// SIMATIC STEP 7 (V5.x) project CAN-O-MAT
// CPU: CPU 314C-2 DP
// station: P_ADR_BUS
// station: Hardware
// station: SIMATIC 300(1)
// program: S7 Program(1)

SYMBOL_TABLE
"FC2"	FC 2	FC 2	// Освещение внутри каномата
"FC3"	FC 3	FC 3	// Блок управления основным приводом
"FC4"	FC 4	FC 4	// Конвеер и подача корпусов
"FC6"	FC 6	FC 6	// Насос смазки (Опция)
"FC7"	FC 7	FC 7	// Смазка сужения
"1-А4"	I 14.1	BOOL	// Кнопки СТОП
"2-S19==2-S22"	I 14.2	BOOL	// Защитное устройство (окна)
"3-М1"	I 14.3	BOOL	// Основной привод включен
"7-Q7"	I 14.5	BOOL	// Автомат защиты насоса смазки банки
"8-Q8"	I 14.6	BOOL	// АВ защиты Кран(опция)
"10-М9а"	I 14.7	BOOL	// Транспорт подачи крышки включен
"РЕЗЕРВ 5"	I 15.0	BOOL	// Внешнее разрешение (или перемычка)
"РЕЗЕРВ 1"	I 15.1	BOOL	// Внешнее разрешение (или перемычка)
"Резерв"	I 15.2	BOOL	// Перемычка
"9-В34"	I 15.5	BOOL	// Опция
"9-В35Е==9-В35S"	I 15.6	BOOL	// Синхронизация выбрасывателя тестовой банки (опция)
"6-Q2"	I 15.7	BOOL	// Автомат защиты масляного насоса
"11-М10а"	I 16.4	BOOL	// Входной транспортер включен
"РЕЗЕРВ 2"	I 16.5	BOOL	// Резерв
"РЕЗЕРВ 3"	I 16.6	BOOL	// Резерв
"5-S11"	I 20.0	BOOL	// Автоматическая работа
"5-S29"	I 20.1	BOOL	// Jog Назад
"ET200S"	I 20.2	BOOL	// Питание подано
"5-S26"	I 20.3	BOOL	// Jog Вперед
"9-S10"	I 20.4	BOOL	// Сжатый воздух
"6-S1"	I 20.5	BOOL	// Давление масла за фильтром
"7-S27"	I 20.6	BOOL	// Наличие давления смазки
"7-S28"	I 20.7	BOOL	// Уровень смазки в бачке
"9-В28"	I 21.0	BOOL	// Датчик увеличения скорости каномата
"9-В29"	I 21.1	BOOL	// Наличие банки(входной конв)
"9-В30"	I 21.2	BOOL	// Датчик затора на выходном конвейере
"3-М1М"	I 21.3	BOOL	// Контроль температур Основного мотора
"9-В10"	I 21.4	BOOL	// Датчик такта
"9-В9"	I 21.5	BOOL	// Входящий запрос
"9-В27"	I 21.6	BOOL	// Опрос выхода
"9-В11"	I 21.7	BOOL	// Станция зауживания
"9-В12"	I 22.0	BOOL	// Станция отбортовки
"9-В13"	I 22.1	BOOL	// Станция зауживания
"9-В14"	I 22.2	BOOL	// Станция закатки №1
"9-В15"	I 22.3	BOOL	// Станция закатки №2
"6-S3"	I 22.6	BOOL	// Импульсы смазки (опция)
"11-B1"	I 22.7	BOOL	// Переполнение входного конвеера
"5-S230"	I 23.0	BOOL	// Кнопка СБРОС
"РЕЗЕРВ 4"	I 23.2	BOOL	// Резерв
"10-В29"	I 23.3	BOOL	// Такт подачи крышки
"10-В30"	I 23.4	BOOL	// Опрос крышки
"10-B31"	I 23.5	BOOL	// Наличие крышки на ленте
"10-В32"	I 23.6	BOOL	// Наличие крышки в магазине
"10-В33"	I 23.7	BOOL	// Наличие крышки
"5-S244"	I 24.4	BOOL	// Основной мотор ВКЛ
"5-S245"	I 24.5	BOOL	// Основной мотор ОТКЛ
"5-S246"	I 24.6	BOOL	// Каномат СТОП Открыт
"5-S247"	I 24.7	BOOL	// Каномат СТОП Закрыт
"М0.0"	M 0.0	BOOL	// Меркер всегда выключ.
"М0.1"	M 0.1	BOOL	// Теплый пуск CPU. Меркер всегда включен
"М0.5"	M 0.5	BOOL	// Меркер всегда выключ.
"М1.0"	M 1.0	BOOL	// Меркер неисправного состояния
"М1.1"	M 1.1	BOOL	// Тригер Основной мотор ВКЛ(Ручн. реж)
"М1.2"	M 1.2	BOOL	// Тригер Основной мотор ВКЛ(Авт. реж)
"М1.3"	M 1.3	BOOL	// Тригер Основной мотор Jog Вперед
"М1.5"	M 1.5	BOOL	// Тригер Основной мотор Jog Назад
"М2.0"	M 2.0	BOOL	// Меркер включения Основного мотора
"М2.2"	M 2.2	BOOL	// Входной конвейер переполнен
"М2.7"	M 2.7	BOOL	// Меркер затора на выходном конвейере
"М3.0"	M 3.0	BOOL	// Тригер включ. конвеера
"М3.3"	M 3.3	BOOL	// Наличие банки на входе
"М4.0"	M 4.0	BOOL	// Тригер включ. освещение каномата
"М6.2"	M 6.2	BOOL	// Меркер включ. масляного насоса для сужения
"М12.0"	M 12.0	BOOL	// Меркер включ. клапана подачи корпусов
"М16.4"	M 16.4	BOOL	// Меркер включения входного транспорт.
"М16.5"	M 16.5	BOOL	// Меркер включения РЕЗЕРВ 9
"М100.3"	M 100.3	BOOL	// Меркер ВКЛ входного транспорт
"М100.4"	M 100.4	BOOL	// РЕЗЕРВ 2,3 Всегда включен
"М100.7"	M 100.7	BOOL	// Входной транспорт. РАБОТАЕТ
"М101.0"	M 101.0	BOOL	// Меркер нормальной работы
"М220.1"	M 220.1	BOOL	// Автомат защиты насоса смазки банки ВЫКЛЮЧЕН
"М220.2"	M 220.2	BOOL	// АВ защиты Кран (опция) ВЫКЛЮЧЕН
"М221.0"	M 221.0	BOOL	// Нажата Аварийная кнопка СТОП
"М221.1"	M 221.1	BOOL	// Защитное устройство ОТКРЫТО
"М221.2"	M 221.2	BOOL	// Меркер контроля выкл. состояния Основного привода
"М221.3"	M 221.3	BOOL	// Меркер контроля температур Основного мотора
"М221.6"	M 221.6	BOOL	// НЕТ давления масла на сужении
"М222.0"	M 222.0	BOOL	// НЕТ крышки в магазине
"М222.3"	M 222.3	BOOL	// НЕТ смазки (опция)
"М222.5"	M 222.5	BOOL	// Синхронизация выбрасывателя тестовой банки (опция)
"М222.6"	M 222.6	BOOL	// Автомат защиты масляного насоса ВЫКЛЮЧЕН
"М223.5"	M 223.5	BOOL	// Каномат остановлен
"М223.7"	M 223.7	BOOL	// Транспорт подачи крышки ВЫКЛЮЧЕН
"М227.7"	M 227.7	BOOL	// Входной транспорт. НЕ РАБОТАЕТ
"М229.0"	M 229.0	BOOL	// Исправная работа
"М229.1"	M 229.1	BOOL	// Затор на выходном конвейере
"М248.2"	M 248.2	BOOL	// Меркер Освещение каномата Выключено
"М249.4"	M 249.4	BOOL	// Входной транспорт. ВЫКЛЮЧЕН
"М249.6"	M 249.6	BOOL	// РЕЗЕРВ 9 ВЫКЛЮЧЕН
"М250.2"	M 250.2	BOOL	// Меркер Освещение каномата Включено
"М251.4"	M 251.4	BOOL	// Входной транспорт. ВКЛЮЧЕН
"М251.6"	M 251.6	BOOL	// РЕЗЕРВ 9 ВКЛЮЧЕН
"3-К1"	Q 14.0	BOOL	// Подача питания на частотные привода
"1-К5"	Q 14.1	BOOL	// Сброс  Перезагрузка
"2-К3"	Q 14.2	BOOL	// Освещение каномата
"3-М1-2"	Q 14.3	BOOL	// Основной мотор (быстрое торможение
"3-M1-3"	Q 14.4	BOOL	// Основной мотор(Jog вперед)
"3-М1-4"	Q 14.5	BOOL	// Основной мотор(Jog назад)
"12-К2"	Q 14.6	BOOL	// Каномат в ожидании
"12-К3"	Q 14.7	BOOL	// Каномат в ожидании
"3-М1-1"	Q 15.0	BOOL	// Основной мотор (ВКЛ)
"12-К1"	Q 15.1	BOOL	// Каномат в работе
"7-K7"	Q 15.2	BOOL	// Масляной насос для сужения
"10-M9"	Q 15.4	BOOL	// Транспортер подачи крышки
"6-К2"	Q 15.5	BOOL	// Насос смазки (Опция)
"9-Y10"	Q 15.6	BOOL	// Опция
"11-М10"	Q 16.4	BOOL	// Входной транспортер
"РЕЗЕРВ 9"	Q 16.5	BOOL	// Резерв
"РЕЗЕРВ 10"	Q 16.6	BOOL	// Резерв
"РЕЗЕРВ 6"	Q 17.5	BOOL	// Резерв
"РЕЗЕРВ 7"	Q 17.6	BOOL	// Резерв
"РЕЗЕРВ 8"	Q 17.7	BOOL	// Резерв
"9-Y3"	Q 20.0	BOOL	// Клапан подачи корпусов
"7-Y5"	Q 20.1	BOOL	// Клапан распыления при сужении
"10-Y14"	Q 20.2	BOOL	// Клапан подачи крышки
"5-Н203"	Q 20.3	BOOL	// Лампа АВАРИЯ
"5-Н206"	Q 20.6	BOOL	// Лампа Основной мотор Включен
"5-Н207"	Q 20.7	BOOL	// Лампа Конвеер Включен
"SET_CLK"	SFC 0	SFC 0	// Set System Clock
"READ_CLK"	SFC 1	SFC 1	// Read System Clock
"SET_RTM"	SFC 2	SFC 2	// Set Run-Time Meter
"CTRL_RTM"	SFC 3	SFC 3	// Start/Stop Run-Time Meter
"READ_RTM"	SFC 4	SFC 4	// Read Run-Time Meter
"BLKMOV"	SFC 20	SFC 20	// Copy Variables
"FILL"	SFC 21	SFC 21	// Initialize a Memory Area
"Т1"	T 1	TIMER	// Задержка выключения 3-К1
"Т2"	T 2	TIMER	// Задержка срабатывания 9-В29 (включ.)
"Т3"	T 3	TIMER	// Таймер включ. на 1 сек. и выключ.
"Т4"	T 4	TIMER	// Задержка срабатывания 9-В29 (отключ.)
"Т11"	T 11	TIMER	// Задержка включения
"Т14"	T 14	TIMER	// Задержка срабатывания датчика 9-В28
"Т15"	T 15	TIMER	// Задержка включения датчика 9-В30 Затор на выходном конв
"Т16"	T 16	TIMER	// Задержка выключен датчика 9-В30 Затор на выходном конв.
"Т22"	T 22	TIMER	// Задержка включ. датчика 11-В1
"Т26"	T 26	TIMER	// Задержка включен. РЕЗЕРВ 5
"Т27"	T 27	TIMER	// Задержка выключен. РЕЗЕРВ 5
"Т28"	T 28	TIMER	// Задержка выключен. РЕЗЕРВ 1
"Т29"	T 29	TIMER	// Задержка включен. РЕЗЕРВ 1
"Т37"	T 37	TIMER	// Задержка отключения
"Т39"	T 39	TIMER	// Задержка включения
"Т40"	T 40	TIMER	// Задержка срабатывания
"Т42"	T 42	TIMER	// Задержка отключ. датчика 11-В1
"Т44"	T 44	TIMER	// Задержка включения "М0.1"
"Т45"	T 45	TIMER	// Таймер отсчитывает время и выключает
"Т46"	T 46	TIMER	// Задержка включения 2-S19=2S22
"Т50"	T 50	TIMER	// Таймер срабатыв. через время после начала тормож. Осн.  мотора
"Т52"	T 52	TIMER	// Задержка срабатыван датчика такта во включ. положении
"Т53"	T 53	TIMER	// Задержка срабатыван датчика такта в отключ. положении
"Т60"	T 60	TIMER	// Время смазки
"Т61"	T 61	TIMER	// Время между смазками
"Т120"	T 120	TIMER	// Задержка включ. клапана подачи корпусов
END_SYMBOL_TABLE

FUNCTION_BLOCK FB 100
AUTHOR : Joehring
VERSION : 0.1
BEGIN
// (block stored without names or comments; labels and parameter names are numbered)
NETWORK
TITLE =
      BLD   7;
      =     L 8.0;
      TAR2  LD 4;
      L     DINO;
      T     LW 9;
      +AR2  P#12.0;
      TAR2;
      LAR2  LD 4;
      T     LD 11;
      UC    "READ_CLK";
      {     P#L 2.0, P#L 9.0 };
      LAR2  LD 4;
      BLD   8;
      NOP   0;
NETWORK
TITLE =
      A(;
      A(;
      L     DIW [AR2,P#0.0];
      L     DIW [AR2,P#2.0];
      ==I;
      );
      =     L 0.0;
      A     L 0.0;
      FP    DIX [AR2,P#42.2];
      JNB   M001;
      L     DID 12;
      T     DID 24;
      SET;
      SAVE;
      CLR;
M001: A     BR;
      );
      JNB   M002;
      L     DID 16;
      T     DID 28;
M002: NOP   0;
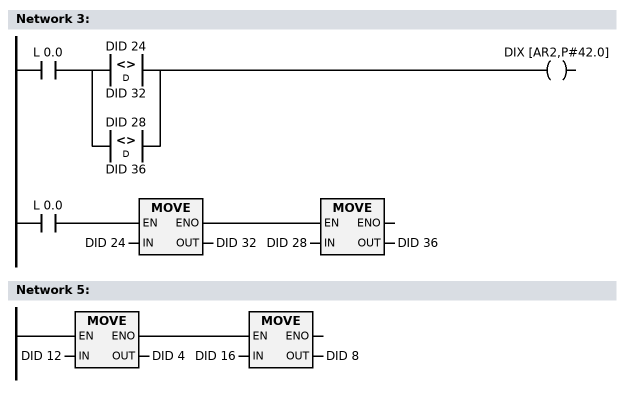
NETWORK
TITLE =
      A     L 0.0;
      =     L 4.0;
      A     L 4.0;
      A(;
      O(;
      L     DID 24;
      L     DID 32;
      <>D;
      );
      O(;
      L     DID 28;
      L     DID 36;
      <>D;
      );
      );
      =     DIX [AR2,P#42.0];
      A(;
      A     L 4.0;
      JNB   M003;
      L     DID 24;
      T     DID 32;
      SET;
      SAVE;
      CLR;
M003: A     BR;
      );
      JNB   M004;
      L     DID 28;
      T     DID 36;
M004: NOP   0;
NETWORK
TITLE =
      A     DIX [AR2,P#42.0];
      FP    DIX [AR2,P#42.1];
      JNB   M005;
      BLD   7;
      =     L 8.0;
      TAR2  LD 4;
      L     DINO;
      T     LW 9;
      +AR2  P#24.0;
      TAR2;
      LAR2  LD 4;
      T     LD 11;
      UC    "SET_CLK";
      {     P#L 9.0, P#L 2.0 };
      LAR2  LD 4;
      BLD   8;
M005: NOP   0;
NETWORK
TITLE =
      A(;
      L     DID 12;
      T     DID 4;
      SET;
      SAVE;
      CLR;
      A     BR;
      );
      JNB   M006;
      L     DID 16;
      T     DID 8;
M006: NOP   0;
END_FUNCTION_BLOCK

// FB 125: know-how protected block, not included

FUNCTION "FC2" : VOID	// FC 2
TITLE = Освещение внутри каномата.
//Включение освещения внутри каномата.
AUTHOR : Stolz
VERSION : 0.1
VAR_TEMP
  TEMP0 : BOOL ;
END_VAR
BEGIN
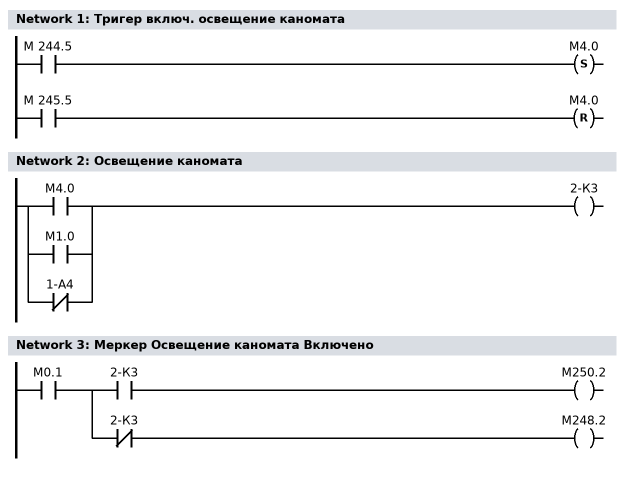
NETWORK
TITLE = Тригер включ. освещение каномата
      A     M 244.5;
      S     "М4.0";
      A     M 245.5;
      R     "М4.0";
      NOP   0;
NETWORK
TITLE = Освещение каномата
      O     "М4.0";
      O     "М1.0";
      ON    "1-А4";
      =     "2-К3";
NETWORK
TITLE = Меркер Освещение каномата Включено
      A     "М0.1";
      =     L 1.0;
      A     L 1.0;
      A     "2-К3";
      =     "М250.2";
      A     L 1.0;
      AN    "2-К3";
      =     "М248.2";
END_FUNCTION

FUNCTION "FC3" : VOID	// FC 3
TITLE = Блок управления основным приводом.
AUTHOR : Stolz
FAMILY : Maschfkt
NAME : Hauptmot
VERSION : 0.1
BEGIN
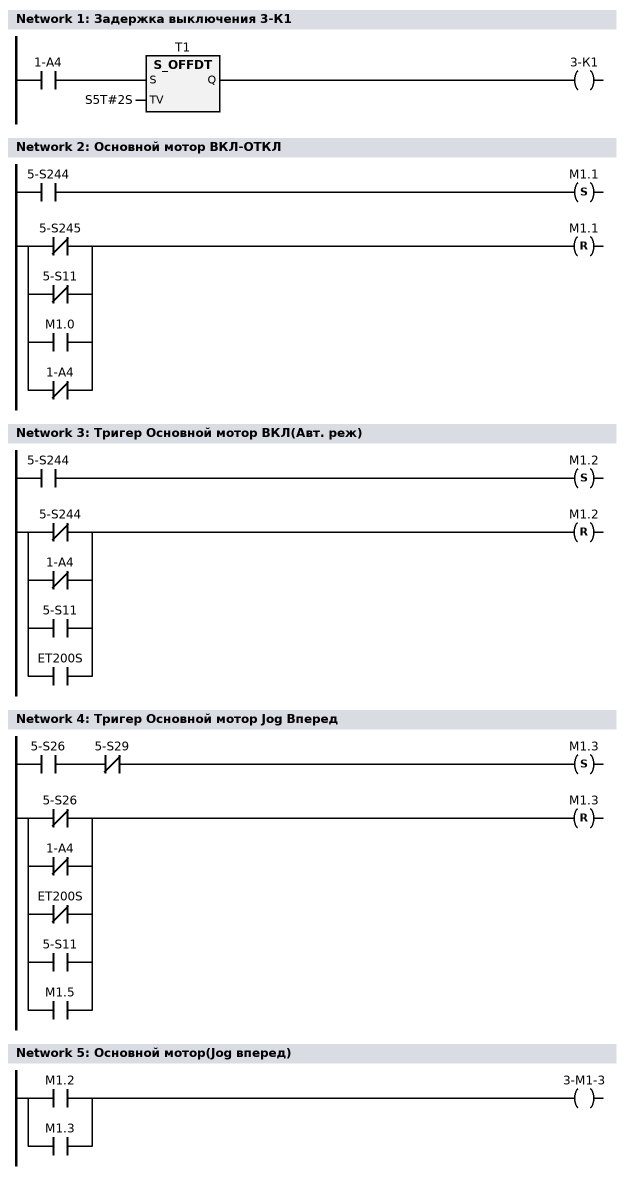
NETWORK
TITLE = Задержка выключения 3-К1
//После нажатия на любую из аварийных кнопок СТОП питание с частотных приводов 
//отключится спустя время, установленное в Т1.
      A     "1-А4";
      L     S5T#2S;
      SF    "Т1";
      NOP   0;
      NOP   0;
      NOP   0;
      A     "Т1";
      =     "3-К1";
NETWORK
TITLE = Основной мотор ВКЛ-ОТКЛ
      A     "5-S244";
      S     "М1.1";
      A(;
      ON    "5-S245";
      ON    "5-S11";
      O     "М1.0";
      ON    "1-А4";
      );
      R     "М1.1";
      NOP   0;
NETWORK
TITLE = Тригер Основной мотор ВКЛ(Авт. реж)
      A     "5-S244";
      S     "М1.2";
      A(;
      ON    "5-S244";
      ON    "1-А4";
      O     "5-S11";
      O     "ET200S";
      );
      R     "М1.2";
      NOP   0;
NETWORK
TITLE = Тригер Основной мотор Jog Вперед
      A     "5-S26";
      AN    "5-S29";
      S     "М1.3";
      A(;
      ON    "5-S26";
      ON    "1-А4";
      ON    "ET200S";
      O     "5-S11";
      O     "М1.5";
      );
      R     "М1.3";
      NOP   0;
NETWORK
TITLE = Основной мотор(Jog вперед)
      O     "М1.2";
      O     "М1.3";
      =     "3-M1-3";
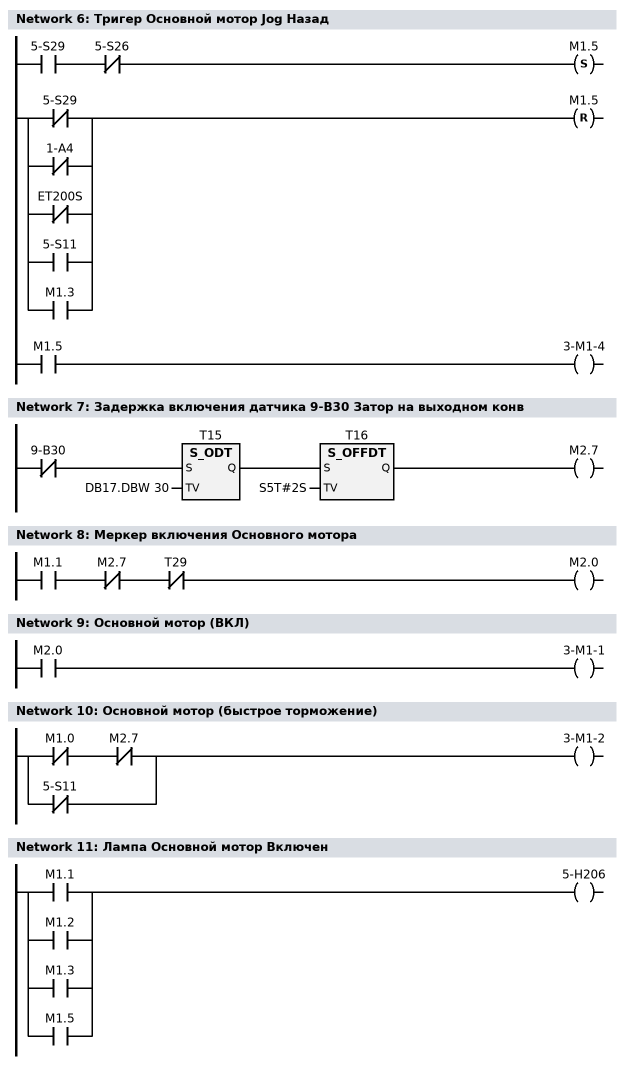
NETWORK
TITLE = Тригер Основной мотор Jog Назад
      A     "5-S29";
      AN    "5-S26";
      S     "М1.5";
      A(;
      ON    "5-S29";
      ON    "1-А4";
      ON    "ET200S";
      O     "5-S11";
      O     "М1.3";
      );
      R     "М1.5";
      A     "М1.5";
      =     "3-М1-4";
NETWORK
TITLE = Задержка включения датчика 9-В30 Затор на выходном конв
      A(;
      AN    "9-В30";
      L     DB17.DBW 30;
      SD    "Т15";
      NOP   0;
      NOP   0;
      NOP   0;
      A     "Т15";
      );
      L     S5T#2S;
      SF    "Т16";
      NOP   0;
      NOP   0;
      NOP   0;
      A     "Т16";
      =     "М2.7";
NETWORK
TITLE = Меркер включения Основного мотора
      A     "М1.1";
      AN    "М2.7";
      AN    "Т29";
      =     "М2.0";
NETWORK
TITLE = Основной мотор (ВКЛ)
      A     "М2.0";
      =     "3-М1-1";
NETWORK
TITLE = Основной мотор (быстрое торможение)
      AN    "М1.0";
      AN    "М2.7";
      ON    "5-S11";
      =     "3-М1-2";
NETWORK
TITLE = Лампа Основной мотор Включен
      O     "М1.1";
      O     "М1.2";
      O     "М1.3";
      O     "М1.5";
      =     "5-Н206";
END_FUNCTION

FUNCTION "FC4" : VOID	// FC 4
TITLE = Конвеер и подача корпусов.
AUTHOR : Stolz
VERSION : 0.1
VAR_TEMP
  TEMP0 : BOOL ;
END_VAR
BEGIN
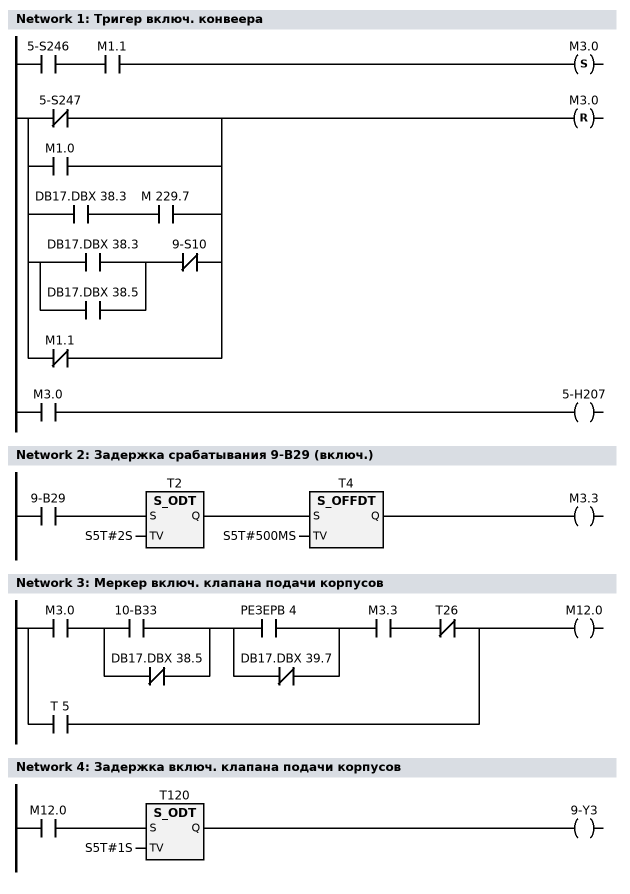
NETWORK
TITLE = Тригер включ. конвеера
      A     "5-S246";
      A     "М1.1";
      S     "М3.0";
      A(;
      ON    "5-S247";
      O     "М1.0";
      O;
      A     DB17.DBX 38.3;
      A     M 229.7;
      O;
      A(;
      O     DB17.DBX 38.3;
      O     DB17.DBX 38.5;
      );
      AN    "9-S10";
      ON    "М1.1";
      );
      R     "М3.0";
      A     "М3.0";
      =     "5-Н207";
NETWORK
TITLE = Задержка срабатывания 9-В29 (включ.)
      A(;
      A     "9-В29";
      L     S5T#2S;
      SD    "Т2";
      NOP   0;
      NOP   0;
      NOP   0;
      A     "Т2";
      );
      L     S5T#500MS;
      SF    "Т4";
      NOP   0;
      NOP   0;
      NOP   0;
      A     "Т4";
      =     "М3.3";
NETWORK
TITLE = Меркер включ. клапана подачи корпусов
      A     "М3.0";
      A(;
      O     "10-В33";
      ON    DB17.DBX 38.5;
      );
      A(;
      O     "РЕЗЕРВ 4";
      ON    DB17.DBX 39.7;
      );
      A     "М3.3";
      AN    "Т26";
      O     T 5;
      =     "М12.0";
NETWORK
TITLE = Задержка включ. клапана подачи корпусов
      A     "М12.0";
      L     S5T#1S;
      SD    "Т120";
      NOP   0;
      NOP   0;
      NOP   0;
      A     "Т120";
      =     "9-Y3";
END_FUNCTION

FUNCTION "FC6" : VOID	// FC 6
TITLE = Включение насоса смазки.
//Включение насоса смазки(Опция)
AUTHOR : Stolz
NAME : Schmier
VERSION : 0.1
BEGIN
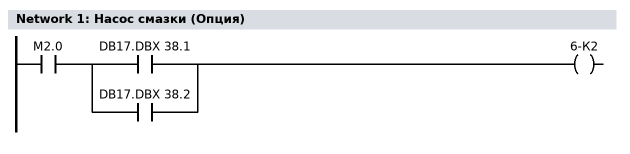
NETWORK
TITLE = Насос смазки (Опция)
      A     "М2.0";
      A(;
      O     DB17.DBX 38.1;
      O     DB17.DBX 38.2;
      );
      =     "6-К2";
END_FUNCTION

FUNCTION "FC7" : VOID	// FC 7
TITLE = Блок управления смазкой сужения.
AUTHOR : Stolz
VERSION : 0.1
BEGIN
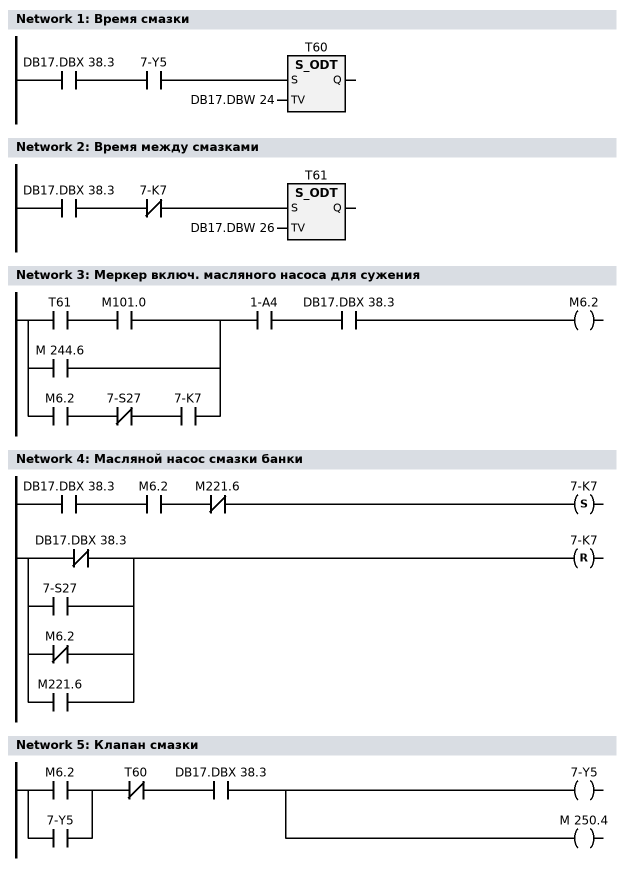
NETWORK
TITLE = Время смазки
      A     DB17.DBX 38.3;
      A     "7-Y5";
      L     DB17.DBW 24;
      SD    "Т60";
      NOP   0;
      NOP   0;
      NOP   0;
      NOP   0;
NETWORK
TITLE = Время между смазками
      A     DB17.DBX 38.3;
      AN    "7-K7";
      L     DB17.DBW 26;
      SD    "Т61";
      NOP   0;
      NOP   0;
      NOP   0;
      NOP   0;
NETWORK
TITLE = Меркер включ. масляного насоса для сужения
      A(;
      A     "Т61";
      A     "М101.0";
      O     M 244.6;
      O;
      A     "М6.2";
      AN    "7-S27";
      A     "7-K7";
      );
      A     "1-А4";
      A     DB17.DBX 38.3;
      =     "М6.2";
NETWORK
TITLE = Масляной насос смазки банки
      A     DB17.DBX 38.3;
      A     "М6.2";
      AN    "М221.6";
      S     "7-K7";
      A(;
      ON    DB17.DBX 38.3;
      O     "7-S27";
      ON    "М6.2";
      O     "М221.6";
      );
      R     "7-K7";
      NOP   0;
NETWORK
TITLE = Клапан смазки
      A(;
      O     "М6.2";
      O     "7-Y5";
      );
      AN    "Т60";
      A     DB17.DBX 38.3;
      =     "7-Y5";
      =     M 250.4;
END_FUNCTION

FUNCTION FC 10 : VOID
AUTHOR : Stolz
NAME : Deckelfi
VERSION : 0.3
VAR_TEMP
  TEMP0 : DWORD ;
  TEMP1 : BOOL ;
  TEMP2 : BOOL ;
  TEMP3 : BOOL ;
END_VAR
BEGIN
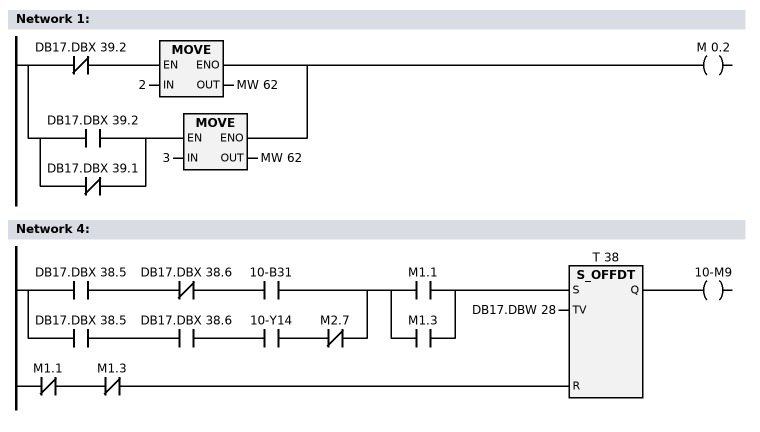
NETWORK
TITLE =
      O(;
      AN    DB17.DBX 39.2;
      JNB   _001;
      L     2;
      T     MW 62;
      SET;
      SAVE;
      CLR;
_001: A     BR;
      );
      O(;
      A(;
      O     DB17.DBX 39.2;
      ON    DB17.DBX 39.1;
      );
      JNB   _002;
      L     3;
      T     MW 62;
      SET;
      SAVE;
      CLR;
_002: A     BR;
      );
      =     M 0.2;
NETWORK
TITLE =
      A(;
      A     M 21.4;
      CD    C 36;
      BLD   101;
      A(;
      O     M 21.7;
      O     "5-S246";
      );
      L     MW 62;
      S     C 36;
      NOP   0;
      NOP   0;
      NOP   0;
      A     C 36;
      );
      NOT;
      =     #TEMP1;
NETWORK
TITLE =
      A(;
      A     M 21.7;
      CD    C 37;
      BLD   101;
      A(;
      O     #TEMP1;
      O     "5-S246";
      );
      L     DB17.DBW 56;
      S     C 37;
      NOP   0;
      NOP   0;
      NOP   0;
      A     C 37;
      );
      NOT;
      A     "9-Y3";
      =     M 1.4;
NETWORK
TITLE =
      A(;
      A     DB17.DBX 38.5;
      AN    DB17.DBX 38.6;
      A     "10-B31";
      O;
      A     DB17.DBX 38.5;
      A     DB17.DBX 38.6;
      A     "10-Y14";
      AN    "М2.7";
      );
      A(;
      O     "М1.1";
      O     "М1.3";
      );
      L     DB17.DBW 28;
      SF    T 38;
      AN    "М1.1";
      AN    "М1.3";
      R     T 38;
      NOP   0;
      NOP   0;
      A     T 38;
      =     "10-M9";
END_FUNCTION

FUNCTION FC 11 : VOID
AUTHOR : Stolz
VERSION : 0.2
BEGIN
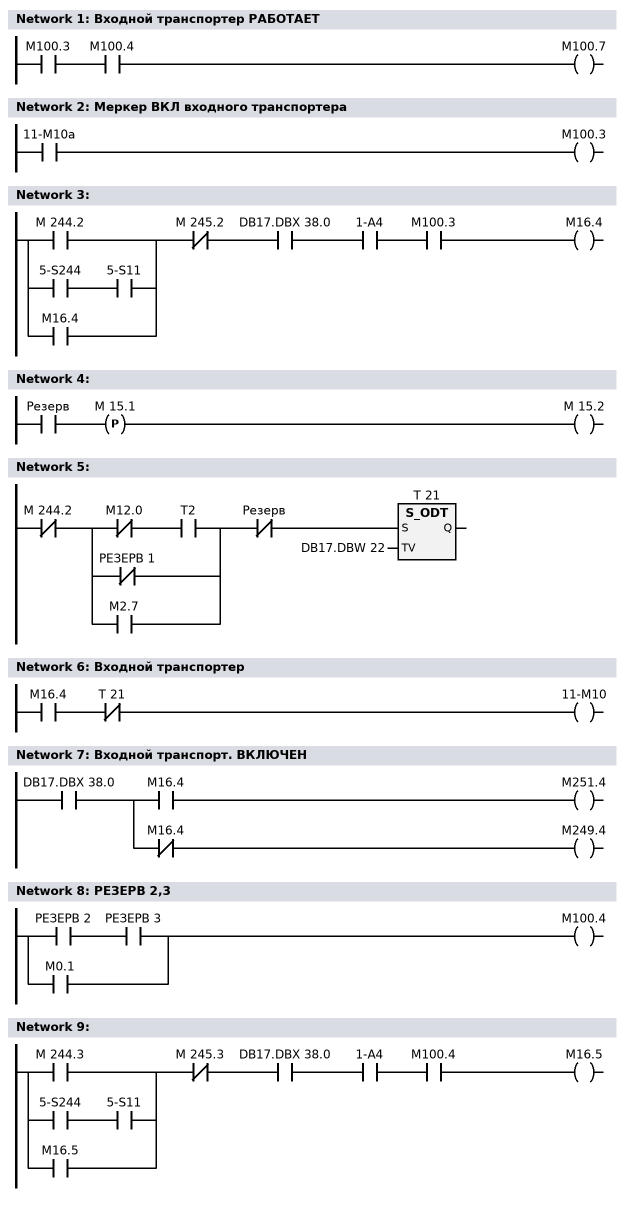
NETWORK
TITLE = Входной транспортер РАБОТАЕТ
      A     "М100.3";
      A     "М100.4";
      =     "М100.7";
NETWORK
TITLE = Меркер ВКЛ входного транспортера
      A     "11-М10а";
      =     "М100.3";
NETWORK
TITLE =
      A(;
      O     M 244.2;
      O;
      A     "5-S244";
      A     "5-S11";
      O     "М16.4";
      );
      AN    M 245.2;
      A     DB17.DBX 38.0;
      A     "1-А4";
      A     "М100.3";
      =     "М16.4";
NETWORK
TITLE =
      A     "Резерв";
      FP    M 15.1;
      =     M 15.2;
NETWORK
TITLE =
      AN    M 244.2;
      A(;
      AN    "М12.0";
      A     "Т2";
      ON    "РЕЗЕРВ 1";
      O     "М2.7";
      );
      AN    "Резерв";
      L     DB17.DBW 22;
      SD    T 21;
      NOP   0;
      NOP   0;
      NOP   0;
      NOP   0;
NETWORK
TITLE = Входной транспортер
      A     "М16.4";
      AN    T 21;
      =     "11-М10";
NETWORK
TITLE = Входной транспорт. ВКЛЮЧЕН
      A     DB17.DBX 38.0;
      =     L 0.0;
      A     L 0.0;
      A     "М16.4";
      =     "М251.4";
      A     L 0.0;
      AN    "М16.4";
      =     "М249.4";
NETWORK
TITLE = РЕЗЕРВ 2,3
      A     "РЕЗЕРВ 2";
      A     "РЕЗЕРВ 3";
      O     "М0.1";
      =     "М100.4";
NETWORK
TITLE =
      A(;
      O     M 244.3;
      O;
      A     "5-S244";
      A     "5-S11";
      O     "М16.5";
      );
      AN    M 245.3;
      A     DB17.DBX 38.0;
      A     "1-А4";
      A     "М100.4";
      =     "М16.5";
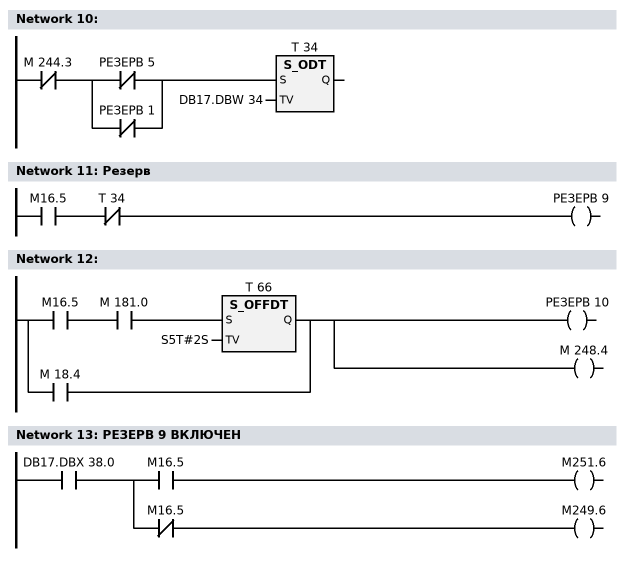
NETWORK
TITLE =
      AN    M 244.3;
      A(;
      ON    "РЕЗЕРВ 5";
      ON    "РЕЗЕРВ 1";
      );
      L     DB17.DBW 34;
      SD    T 34;
      NOP   0;
      NOP   0;
      NOP   0;
      NOP   0;
NETWORK
TITLE = Резерв
      A     "М16.5";
      AN    T 34;
      =     "РЕЗЕРВ 9";
NETWORK
TITLE =
      O(;
      A     "М16.5";
      A     M 181.0;
      L     S5T#2S;
      SF    T 66;
      NOP   0;
      NOP   0;
      NOP   0;
      A     T 66;
      );
      O     M 18.4;
      =     "РЕЗЕРВ 10";
      =     M 248.4;
NETWORK
TITLE = РЕЗЕРВ 9 ВКЛЮЧЕН
      A     DB17.DBX 38.0;
      =     L 0.0;
      A     L 0.0;
      A     "М16.5";
      =     "М251.6";
      A     L 0.0;
      AN    "М16.5";
      =     "М249.6";
END_FUNCTION

FUNCTION FC 12 : VOID
AUTHOR : Stolz
VERSION : 0.3
VAR_TEMP
  TEMP0 : DWORD ;
END_VAR
BEGIN
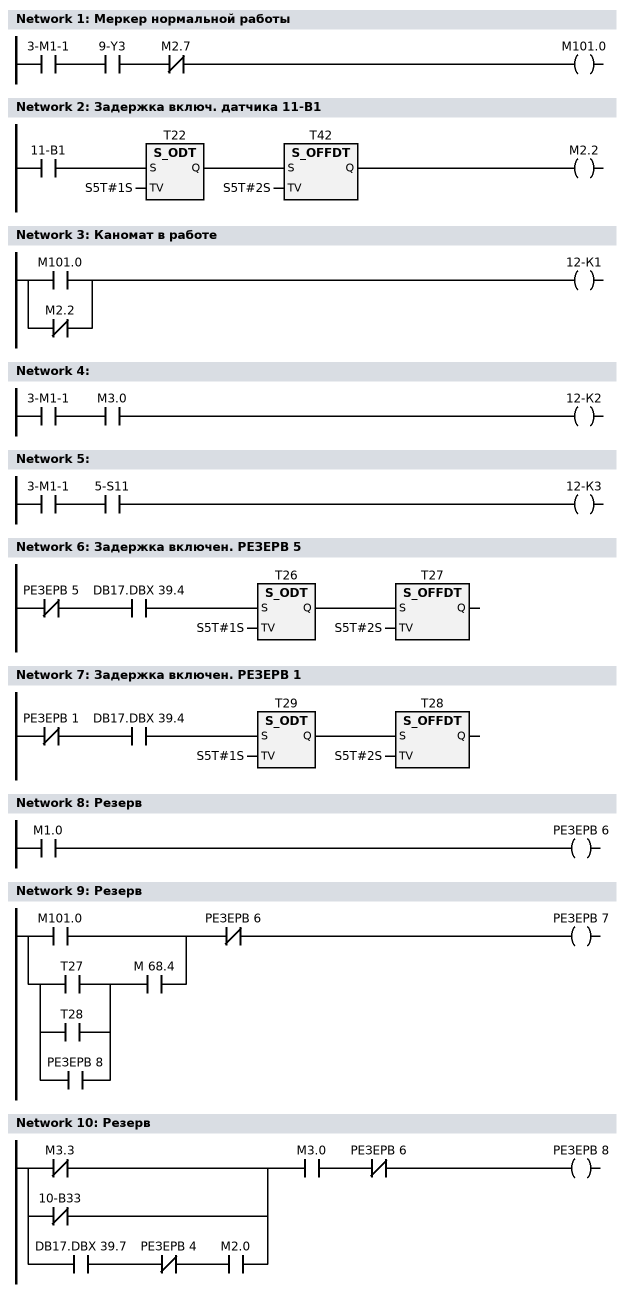
NETWORK
TITLE = Меркер нормальной работы
//Корпуса идут, банка на выходе идет нормально.
      A     "3-М1-1";
      A     "9-Y3";
      AN    "М2.7";
      =     "М101.0";
NETWORK
TITLE = Задержка включ. датчика 11-В1
      A(;
      A     "11-B1";
      L     S5T#1S;
      SD    "Т22";
      NOP   0;
      NOP   0;
      NOP   0;
      A     "Т22";
      );
      L     S5T#2S;
      SF    "Т42";
      NOP   0;
      NOP   0;
      NOP   0;
      A     "Т42";
      =     "М2.2";
NETWORK
TITLE = Каномат в работе
      O     "М101.0";
      ON    "М2.2";
      =     "12-К1";
NETWORK
TITLE =
      A     "3-М1-1";
      A     "М3.0";
      =     "12-К2";
NETWORK
TITLE =
      A     "3-М1-1";
      A     "5-S11";
      =     "12-К3";
NETWORK
TITLE = Задержка включен. РЕЗЕРВ 5
      A(;
      AN    "РЕЗЕРВ 5";
      A     DB17.DBX 39.4;
      L     S5T#1S;
      SD    "Т26";
      NOP   0;
      NOP   0;
      NOP   0;
      A     "Т26";
      );
      L     S5T#2S;
      SF    "Т27";
      NOP   0;
      NOP   0;
      NOP   0;
      NOP   0;
NETWORK
TITLE = Задержка включен. РЕЗЕРВ 1
      A(;
      AN    "РЕЗЕРВ 1";
      A     DB17.DBX 39.4;
      L     S5T#1S;
      SD    "Т29";
      NOP   0;
      NOP   0;
      NOP   0;
      A     "Т29";
      );
      L     S5T#2S;
      SF    "Т28";
      NOP   0;
      NOP   0;
      NOP   0;
      NOP   0;
NETWORK
TITLE = Резерв
      A     "М1.0";
      =     "РЕЗЕРВ 6";
NETWORK
TITLE = Резерв
      A(;
      O     "М101.0";
      O;
      A(;
      O     "Т27";
      O     "Т28";
      O     "РЕЗЕРВ 8";
      );
      A     M 68.4;
      );
      AN    "РЕЗЕРВ 6";
      =     "РЕЗЕРВ 7";
NETWORK
TITLE = Резерв
      A(;
      ON    "М3.3";
      ON    "10-В33";
      O;
      A     DB17.DBX 39.7;
      AN    "РЕЗЕРВ 4";
      A     "М2.0";
      );
      A     "М3.0";
      AN    "РЕЗЕРВ 6";
      =     "РЕЗЕРВ 8";
END_FUNCTION

FUNCTION FC 23 : VOID
AUTHOR : Stolz
VERSION : 0.2
VAR_TEMP
  TEMP0 : DINT ;
  TEMP1 : DINT ;
  TEMP2 : BOOL ;
  TEMP3 : BOOL ;
  TEMP4 : BOOL ;
  TEMP5 : BOOL ;
END_VAR
BEGIN
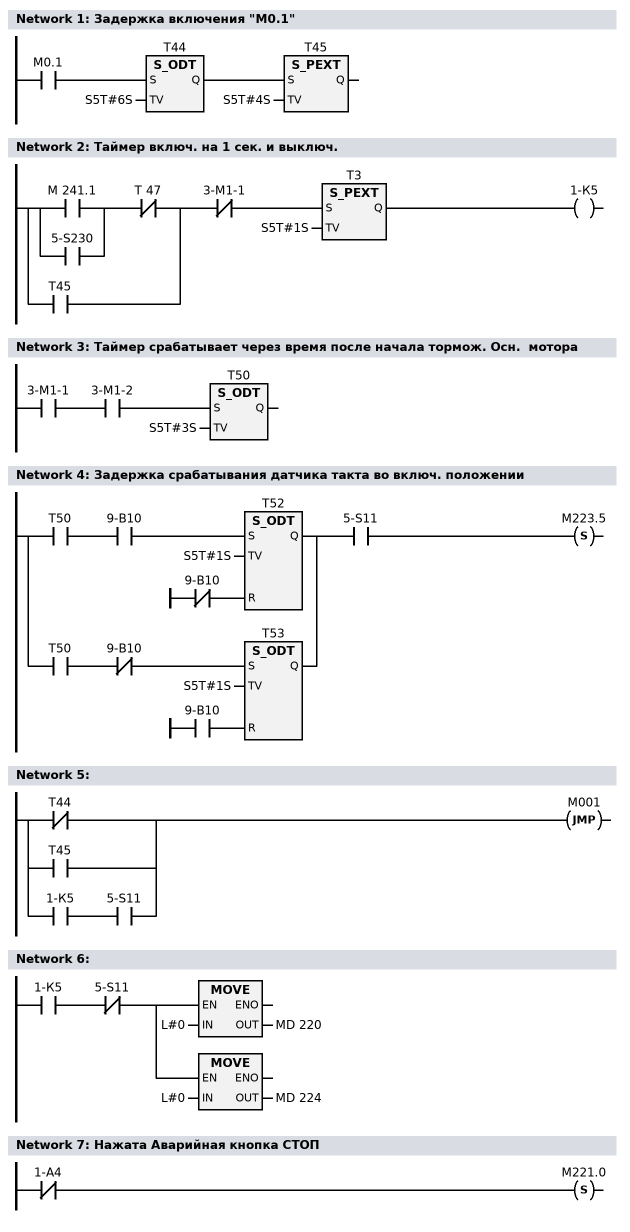
NETWORK
TITLE = Задержка включения "М0.1"
//Т44 включается через 6 сек. после подачи питания на каномат, Т45 включается 
//сразу после срабатывания Т44 и выключается через 4 сек. Остается выключенным до 
//конца работы.
      A(;
      A     "М0.1";
      L     S5T#6S;
      SD    "Т44";
      NOP   0;
      NOP   0;
      NOP   0;
      A     "Т44";
      );
      L     S5T#4S;
      SE    "Т45";
      NOP   0;
      NOP   0;
      NOP   0;
      NOP   0;
NETWORK
TITLE = Таймер включ. на 1 сек. и выключ.
      A(;
      A(;
      O     M 241.1;
      O     "5-S230";
      );
      AN    T 47;
      O     "Т45";
      );
      AN    "3-М1-1";
      L     S5T#1S;
      SE    "Т3";
      NOP   0;
      NOP   0;
      NOP   0;
      A     "Т3";
      =     "1-К5";
NETWORK
TITLE = Таймер срабатывает через время после начала тормож. Осн.  мотора
      A     "3-М1-1";
      A     "3-М1-2";
      L     S5T#3S;
      SD    "Т50";
      NOP   0;
      NOP   0;
      NOP   0;
      NOP   0;
NETWORK
TITLE = Задержка срабатывания датчика такта во включ. положении
      A(;
      O(;
      A     "Т50";
      A     "9-В10";
      L     S5T#1S;
      SD    "Т52";
      AN    "9-В10";
      R     "Т52";
      NOP   0;
      NOP   0;
      A     "Т52";
      );
      O(;
      A     "Т50";
      AN    "9-В10";
      L     S5T#1S;
      SD    "Т53";
      A     "9-В10";
      R     "Т53";
      NOP   0;
      NOP   0;
      A     "Т53";
      );
      );
      A     "5-S11";
      S     "М223.5";
NETWORK
TITLE =
      ON    "Т44";
      O     "Т45";
      O;
      A     "1-К5";
      A     "5-S11";
      JC    M001;
NETWORK
TITLE =
      A     "1-К5";
      AN    "5-S11";
      =     L 9.0;
      A     L 9.0;
      JNB   _001;
      L     L#0;
      T     MD 220;
_001: NOP   0;
      A     L 9.0;
      JNB   _002;
      L     L#0;
      T     MD 224;
_002: NOP   0;
NETWORK
TITLE = Нажата Аварийная кнопка СТОП
      AN    "1-А4";
      S     "М221.0";
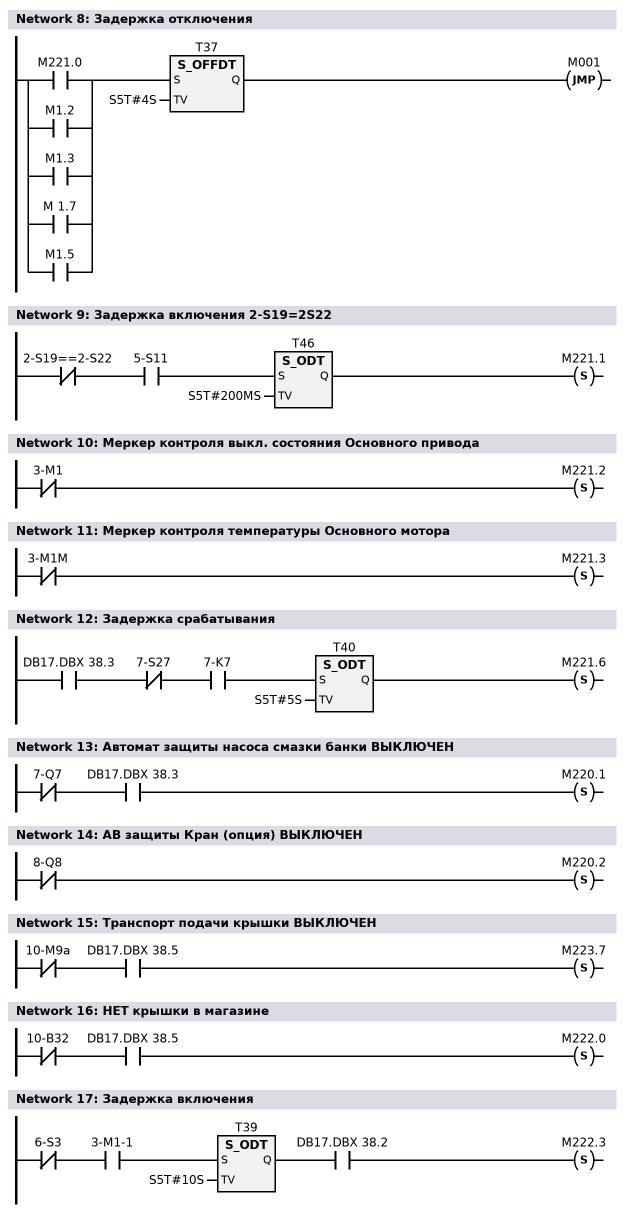
NETWORK
TITLE = Задержка отключения
      A(;
      O     "М221.0";
      O     "М1.2";
      O     "М1.3";
      O     M 1.7;
      O     "М1.5";
      );
      L     S5T#4S;
      SF    "Т37";
      NOP   0;
      NOP   0;
      NOP   0;
      A     "Т37";
      JC    M001;
NETWORK
TITLE = Задержка включения 2-S19=2S22
      AN    "2-S19==2-S22";
      A     "5-S11";
      L     S5T#200MS;
      SD    "Т46";
      NOP   0;
      NOP   0;
      NOP   0;
      A     "Т46";
      S     "М221.1";
NETWORK
TITLE = Меркер контроля выкл. состояния Основного привода
      AN    "3-М1";
      S     "М221.2";
NETWORK
TITLE = Меркер контроля температуры Основного мотора
      AN    "3-М1М";
      S     "М221.3";
NETWORK
TITLE = Задержка срабатывания
      A     DB17.DBX 38.3;
      AN    "7-S27";
      A     "7-K7";
      L     S5T#5S;
      SD    "Т40";
      NOP   0;
      NOP   0;
      NOP   0;
      A     "Т40";
      S     "М221.6";
NETWORK
TITLE = Автомат защиты насоса смазки банки ВЫКЛЮЧЕН
      AN    "7-Q7";
      A     DB17.DBX 38.3;
      S     "М220.1";
NETWORK
TITLE = АВ защиты Кран (опция) ВЫКЛЮЧЕН
      AN    "8-Q8";
      S     "М220.2";
NETWORK
TITLE = Транспорт подачи крышки ВЫКЛЮЧЕН
      AN    "10-М9а";
      A     DB17.DBX 38.5;
      S     "М223.7";
NETWORK
TITLE = НЕТ крышки в магазине
      AN    "10-В32";
      A     DB17.DBX 38.5;
      S     "М222.0";
NETWORK
TITLE = Задержка включения
      A(;
      AN    "6-S3";
      A     "3-М1-1";
      L     S5T#10S;
      SD    "Т39";
      NOP   0;
      NOP   0;
      NOP   0;
      A     "Т39";
      );
      A     DB17.DBX 38.2;
      S     "М222.3";
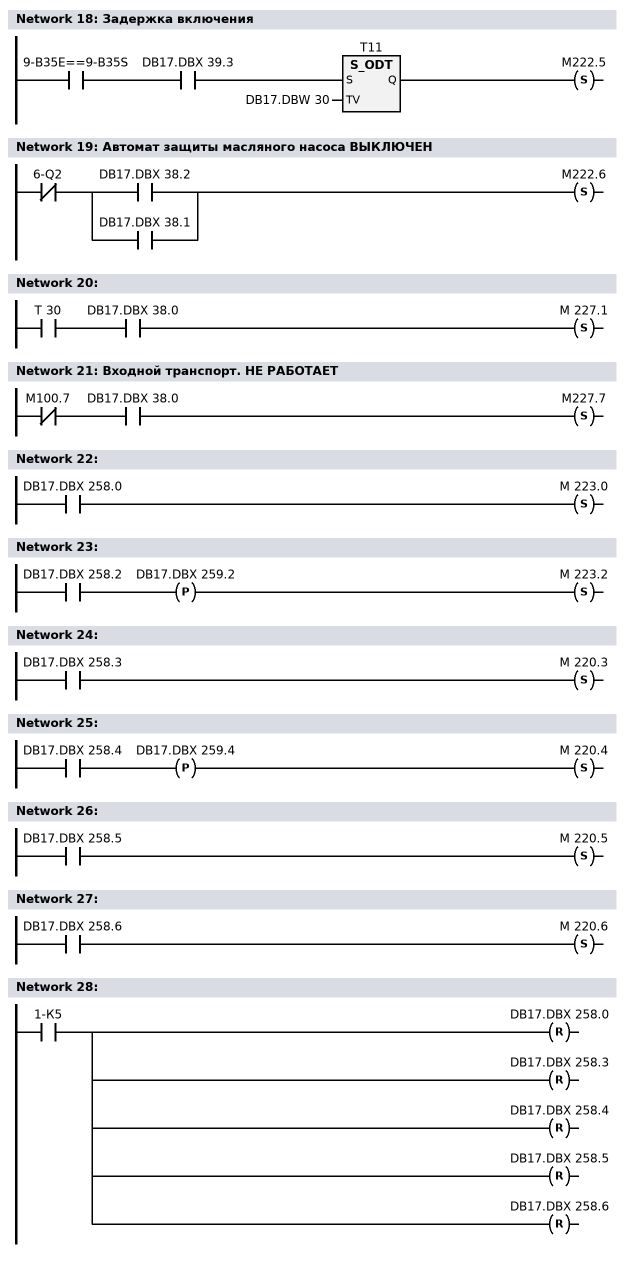
NETWORK
TITLE = Задержка включения
      A     "9-В35Е==9-В35S";
      A     DB17.DBX 39.3;
      L     DB17.DBW 30;
      SD    "Т11";
      NOP   0;
      NOP   0;
      NOP   0;
      A     "Т11";
      S     "М222.5";
NETWORK
TITLE = Автомат защиты масляного насоса ВЫКЛЮЧЕН
      AN    "6-Q2";
      A(;
      O     DB17.DBX 38.2;
      O     DB17.DBX 38.1;
      );
      S     "М222.6";
NETWORK
TITLE =
      A     T 30;
      A     DB17.DBX 38.0;
      S     M 227.1;
NETWORK
TITLE = Входной транспорт. НЕ РАБОТАЕТ
      AN    "М100.7";
      A     DB17.DBX 38.0;
      S     "М227.7";
NETWORK
TITLE =
      A     DB17.DBX 258.0;
      S     M 223.0;
NETWORK
TITLE =
      A     DB17.DBX 258.2;
      FP    DB17.DBX 259.2;
      S     M 223.2;
NETWORK
TITLE =
      A     DB17.DBX 258.3;
      S     M 220.3;
NETWORK
TITLE =
      A     DB17.DBX 258.4;
      FP    DB17.DBX 259.4;
      S     M 220.4;
NETWORK
TITLE =
      A     DB17.DBX 258.5;
      S     M 220.5;
NETWORK
TITLE =
      A     DB17.DBX 258.6;
      S     M 220.6;
NETWORK
TITLE =
      A     "1-К5";
      R     DB17.DBX 258.0;
      R     DB17.DBX 258.3;
      R     DB17.DBX 258.4;
      R     DB17.DBX 258.5;
      R     DB17.DBX 258.6;
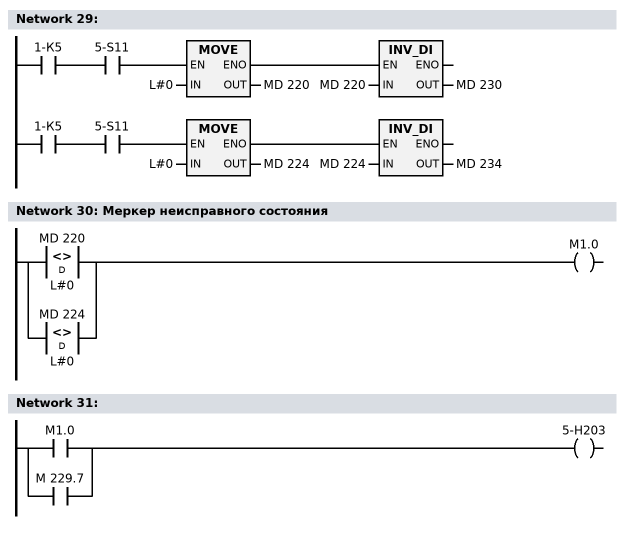
NETWORK
TITLE =
M001: A     "1-К5";
      A     "5-S11";
      =     L 9.0;
      A(;
      A     L 9.0;
      JNB   _003;
      L     L#0;
      T     MD 220;
      SET;
      SAVE;
      CLR;
_003: A     BR;
      );
      JNB   _004;
      L     MD 220;
      INVD;
      T     MD 230;
_004: NOP   0;
      A(;
      A     L 9.0;
      JNB   _005;
      L     L#0;
      T     MD 224;
      SET;
      SAVE;
      CLR;
_005: A     BR;
      );
      JNB   _006;
      L     MD 224;
      INVD;
      T     MD 234;
_006: NOP   0;
NETWORK
TITLE = Меркер неисправного состояния
      O(;
      L     MD 220;
      L     L#0;
      <>D;
      );
      O(;
      L     MD 224;
      L     L#0;
      <>D;
      );
      =     "М1.0";
NETWORK
TITLE =
      O     "М1.0";
      O     M 229.7;
      =     "5-Н203";
END_FUNCTION

FUNCTION FC 24 : VOID
AUTHOR : Stolz
VERSION : 0.2
BEGIN
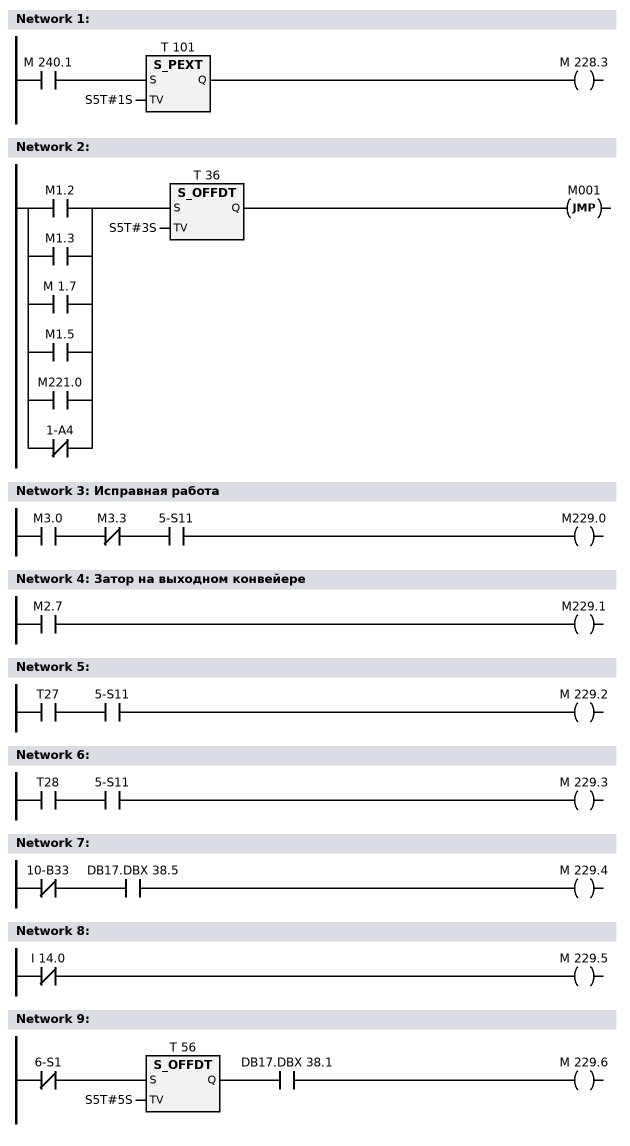
NETWORK
TITLE =
      A     M 240.1;
      L     S5T#1S;
      SE    T 101;
      NOP   0;
      NOP   0;
      NOP   0;
      A     T 101;
      =     M 228.3;
NETWORK
TITLE =
      A(;
      O     "М1.2";
      O     "М1.3";
      O     M 1.7;
      O     "М1.5";
      O     "М221.0";
      ON    "1-А4";
      );
      L     S5T#3S;
      SF    T 36;
      NOP   0;
      NOP   0;
      NOP   0;
      A     T 36;
      JC    M001;
NETWORK
TITLE = Исправная работа
      A     "М3.0";
      AN    "М3.3";
      A     "5-S11";
      =     "М229.0";
NETWORK
TITLE = Затор на выходном конвейере
      A     "М2.7";
      =     "М229.1";
NETWORK
TITLE =
      A     "Т27";
      A     "5-S11";
      =     M 229.2;
NETWORK
TITLE =
      A     "Т28";
      A     "5-S11";
      =     M 229.3;
NETWORK
TITLE =
      AN    "10-В33";
      A     DB17.DBX 38.5;
      =     M 229.4;
NETWORK
TITLE =
      AN    I 14.0;
      =     M 229.5;
NETWORK
TITLE =
      A(;
      AN    "6-S1";
      L     S5T#5S;
      SF    T 56;
      NOP   0;
      NOP   0;
      NOP   0;
      A     T 56;
      );
      A     DB17.DBX 38.1;
      =     M 229.6;
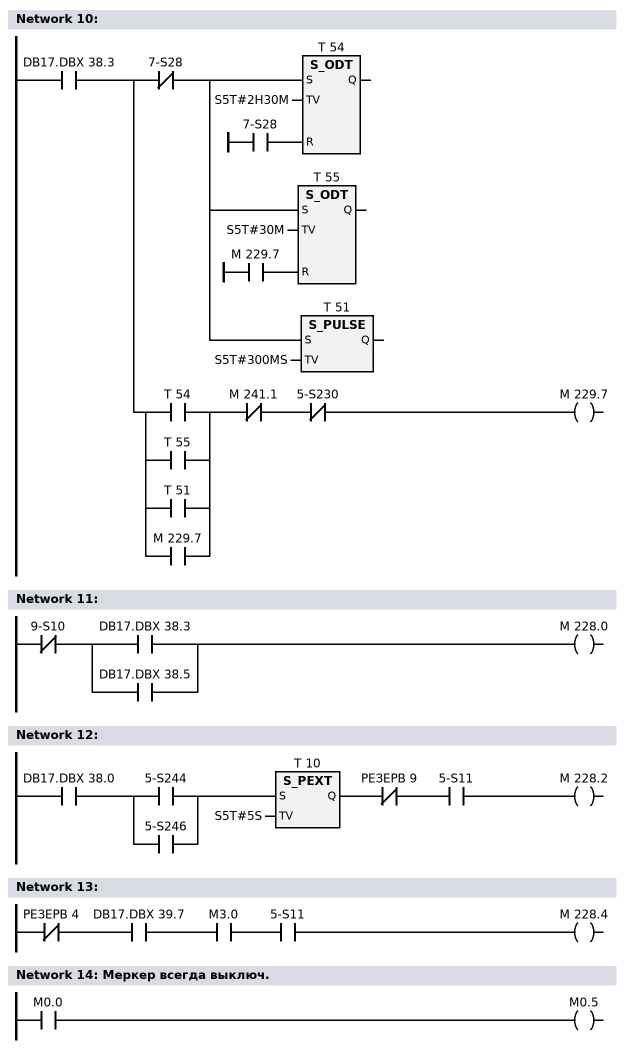
NETWORK
TITLE =
      A     DB17.DBX 38.3;
      =     L 0.0;
      A     L 0.0;
      AN    "7-S28";
      =     L 0.1;
      A     L 0.1;
      L     S5T#2H30M;
      SD    T 54;
      A     "7-S28";
      R     T 54;
      NOP   0;
      NOP   0;
      NOP   0;
      A     L 0.1;
      L     S5T#30M;
      SD    T 55;
      A     M 229.7;
      R     T 55;
      NOP   0;
      NOP   0;
      NOP   0;
      A     L 0.1;
      L     S5T#300MS;
      SP    T 51;
      NOP   0;
      NOP   0;
      NOP   0;
      NOP   0;
      A     L 0.0;
      A(;
      O     T 54;
      O     T 55;
      O     T 51;
      O     M 229.7;
      );
      AN    M 241.1;
      AN    "5-S230";
      =     M 229.7;
NETWORK
TITLE =
      AN    "9-S10";
      A(;
      O     DB17.DBX 38.3;
      O     DB17.DBX 38.5;
      );
      =     M 228.0;
NETWORK
TITLE =
      A(;
      A     DB17.DBX 38.0;
      A(;
      O     "5-S244";
      O     "5-S246";
      );
      L     S5T#5S;
      SE    T 10;
      NOP   0;
      NOP   0;
      NOP   0;
      A     T 10;
      );
      AN    "РЕЗЕРВ 9";
      A     "5-S11";
      =     M 228.2;
NETWORK
TITLE =
      AN    "РЕЗЕРВ 4";
      A     DB17.DBX 39.7;
      A     "М3.0";
      A     "5-S11";
      =     M 228.4;
NETWORK
TITLE = Меркер всегда выключ.
M001: A     "М0.0";
      =     "М0.5";
END_FUNCTION

FUNCTION FC 50 : VOID
AUTHOR : Stolz
VERSION : 0.2
BEGIN
// (block stored without names or comments; labels and parameter names are numbered)
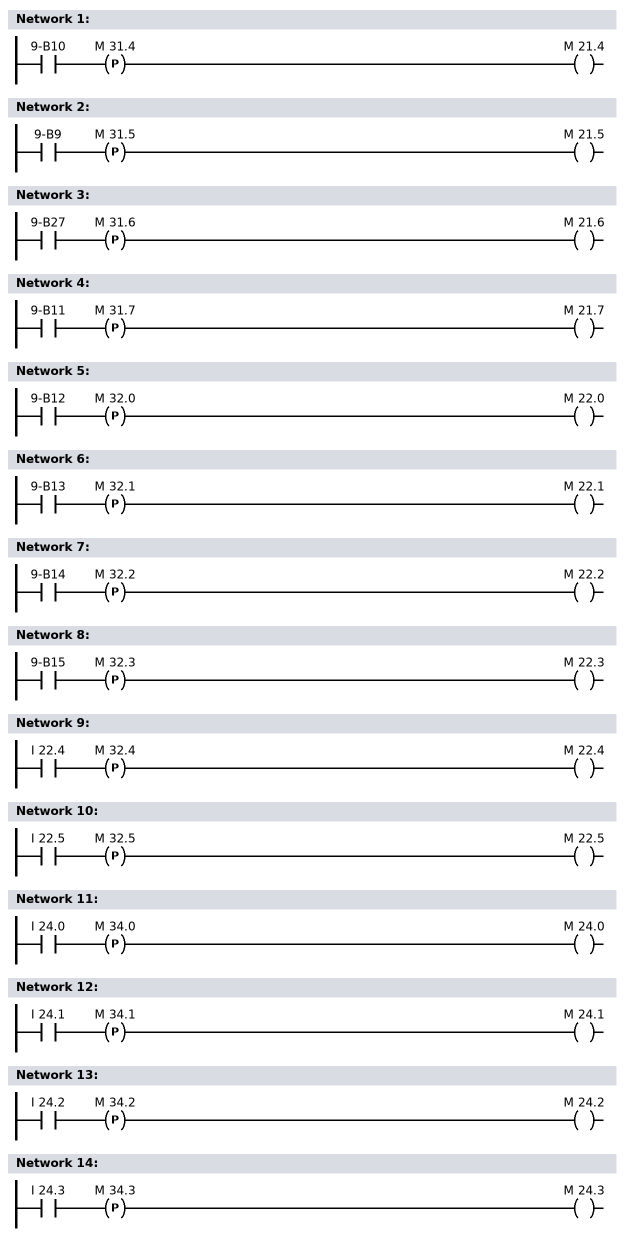
NETWORK
TITLE =
      A     "9-В10";
      FP    M 31.4;
      =     M 21.4;
NETWORK
TITLE =
      A     "9-В9";
      FP    M 31.5;
      =     M 21.5;
NETWORK
TITLE =
      A     "9-В27";
      FP    M 31.6;
      =     M 21.6;
NETWORK
TITLE =
      A     "9-В11";
      FP    M 31.7;
      =     M 21.7;
NETWORK
TITLE =
      A     "9-В12";
      FP    M 32.0;
      =     M 22.0;
NETWORK
TITLE =
      A     "9-В13";
      FP    M 32.1;
      =     M 22.1;
NETWORK
TITLE =
      A     "9-В14";
      FP    M 32.2;
      =     M 22.2;
NETWORK
TITLE =
      A     "9-В15";
      FP    M 32.3;
      =     M 22.3;
NETWORK
TITLE =
      A     I 22.4;
      FP    M 32.4;
      =     M 22.4;
NETWORK
TITLE =
      A     I 22.5;
      FP    M 32.5;
      =     M 22.5;
NETWORK
TITLE =
      A     I 24.0;
      FP    M 34.0;
      =     M 24.0;
NETWORK
TITLE =
      A     I 24.1;
      FP    M 34.1;
      =     M 24.1;
NETWORK
TITLE =
      A     I 24.2;
      FP    M 34.2;
      =     M 24.2;
NETWORK
TITLE =
      A     I 24.3;
      FP    M 34.3;
      =     M 24.3;
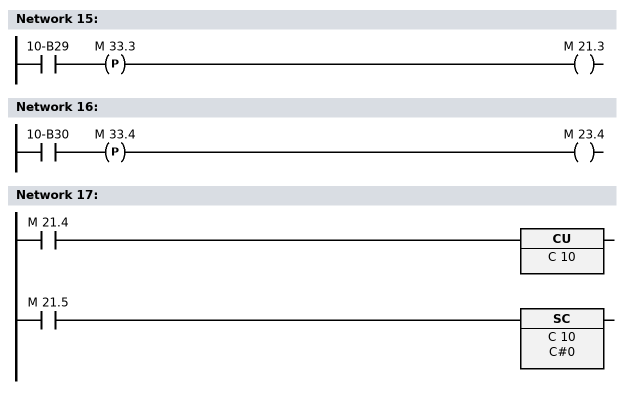
NETWORK
TITLE =
      A     "10-В29";
      FP    M 33.3;
      =     M 21.3;
NETWORK
TITLE =
      A     "10-В30";
      FP    M 33.4;
      =     M 23.4;
NETWORK
TITLE =
      A     M 21.4;
      CU    C 10;
      NOP   0;
      A     M 21.5;
      L     C#0;
      S     C 10;
      NOP   0;
      NOP   0;
      NOP   0;
      NOP   0;
END_FUNCTION

FUNCTION FC 60 : VOID
AUTHOR : Stolz
VERSION : 0.2
BEGIN
// (block stored without names or comments; labels and parameter names are numbered)
NETWORK
TITLE =
      O     "3-М1-1";
      O     "3-M1-3";
      O     "3-М1-4";
      L     S5T#5S;
      SF    T 8;
      A     T 8;
      JC    M001;
      L     0;
      T     MW 10;
      JU    M029;
M001: L     L#1600;
      L     DB17.DBD 138;
      +     L#1600;
      ==D;
      JC    M003;
      T     LD 0;
      A     M 21.7;
      A     M 10.0;
      R     M 10.0;
      JC    M003;
      A     M 21.7;
      AN    M 10.0;
      AN    M 21.4;
      S     M [LD 0];
      JC    M003;
      A     M 21.4;
      A     M 10.0;
      AN    M 21.7;
      JCN   M002;
      L     DB17.DBW 106;
      +     1792;
      ITD;
      T     LD 4;
      S     M [LD 4];
      R     M 10.0;
      R     M [LD 0];
      JU    M003;
M002: A     M 21.7;
      A     M 21.4;
      AN    M 10.0;
      S     M 28.0;
M003: L     L#1600;
      L     DB17.DBD 142;
      +     L#1600;
      ==D;
      JC    M005;
      T     LD 0;
      A     M 22.0;
      A     M 10.1;
      R     M 10.1;
      JC    M005;
      A     M 22.0;
      AN    M 10.1;
      AN    M 21.4;
      S     M [LD 0];
      JC    M005;
      A     M 21.4;
      A     M 10.1;
      AN    M 22.0;
      JCN   M004;
      L     DB17.DBW 108;
      +     1792;
      ITD;
      T     LD 4;
      S     M [LD 4];
      R     M 10.1;
      R     M [LD 0];
      JU    M005;
M004: A     M 22.0;
      A     M 21.4;
      AN    M 10.1;
      S     M 28.1;
M005: L     L#1600;
      L     DB17.DBD 146;
      +     L#1600;
      ==D;
      JC    M007;
      T     LD 0;
      A     M 22.1;
      A     M 10.2;
      R     M 10.2;
      JC    M007;
      A     M 22.1;
      AN    M 10.2;
      AN    M 21.4;
      S     M [LD 0];
      JC    M007;
      A     M 21.4;
      A     M 10.2;
      AN    M 22.1;
      JCN   M006;
      L     DB17.DBW 110;
      +     1792;
      ITD;
      T     LD 4;
      S     M [LD 4];
      R     M 10.2;
      R     M [LD 0];
      JU    M007;
M006: A     M 22.1;
      A     M 21.4;
      AN    M 10.2;
      S     M 28.2;
M007: L     L#1600;
      L     DB17.DBD 150;
      +     L#1600;
      ==D;
      JC    M009;
      T     LD 0;
      A     M 22.2;
      A     M 10.3;
      R     M 10.3;
      JC    M009;
      A     M 22.2;
      AN    M 10.3;
      AN    M 21.4;
      S     M [LD 0];
      JC    M009;
      A     M 21.4;
      A     M 10.3;
      AN    M 22.2;
      JCN   M008;
      L     DB17.DBW 112;
      +     1792;
      ITD;
      T     LD 4;
      S     M [LD 4];
      R     M 10.3;
      R     M [LD 0];
      JU    M009;
M008: A     M 22.2;
      A     M 21.4;
      AN    M 10.3;
      S     M 28.3;
M009: L     L#1600;
      L     DB17.DBD 154;
      +     L#1600;
      ==D;
      JC    M011;
      T     LD 0;
      A     M 22.3;
      A     M 10.4;
      R     M 10.4;
      JC    M011;
      A     M 22.3;
      AN    M 10.4;
      AN    M 21.4;
      S     M [LD 0];
      JC    M011;
      A     M 21.4;
      A     M 10.4;
      AN    M 22.3;
      JCN   M010;
      L     DB17.DBW 114;
      +     1792;
      ITD;
      T     LD 4;
      S     M [LD 4];
      R     M 10.4;
      R     M [LD 0];
      JU    M011;
M010: A     M 22.3;
      A     M 21.4;
      AN    M 10.4;
      S     M 28.4;
M011: L     L#1600;
      L     DB17.DBD 158;
      +     L#1600;
      ==D;
      JC    M013;
      T     LD 0;
      A     M 22.4;
      A     M 10.5;
      R     M 10.5;
      JC    M013;
      A     M 22.4;
      AN    M 10.5;
      AN    M 21.4;
      S     M [LD 0];
      JC    M013;
      A     M 21.4;
      A     M 10.5;
      AN    M 22.4;
      JCN   M012;
      L     DB17.DBW 116;
      +     1792;
      ITD;
      T     LD 4;
      S     M [LD 4];
      R     M 10.5;
      R     M [LD 0];
      JU    M013;
M012: A     M 22.4;
      A     M 21.4;
      AN    M 10.5;
      S     M 28.5;
M013: L     L#1600;
      L     DB17.DBD 162;
      +     L#1600;
      ==D;
      JC    M015;
      T     LD 0;
      A     M 22.5;
      A     M 10.6;
      R     M 10.6;
      JC    M015;
      A     M 22.5;
      AN    M 10.6;
      AN    M 21.4;
      S     M [LD 0];
      JC    M015;
      A     M 21.4;
      A     M 10.6;
      AN    M 22.5;
      JCN   M014;
      L     DB17.DBW 118;
      +     1792;
      ITD;
      T     LD 4;
      S     M [LD 4];
      R     M 10.6;
      R     M [LD 0];
      JU    M015;
M014: A     M 22.5;
      A     M 21.4;
      AN    M 10.6;
      S     M 28.6;
M015: L     L#1600;
      L     DB17.DBD 166;
      +     L#1600;
      ==D;
      JC    M017;
      T     LD 0;
      A     M 24.0;
      A     M 11.0;
      R     M 11.0;
      JC    M017;
      A     M 24.0;
      AN    M 11.0;
      AN    M 21.4;
      S     M [LD 0];
      JC    M017;
      A     M 21.4;
      A     M 11.0;
      AN    M 24.0;
      JCN   M016;
      L     DB17.DBW 120;
      +     1792;
      ITD;
      T     LD 4;
      S     M [LD 4];
      R     M 11.0;
      R     M [LD 0];
      JU    M017;
M016: A     M 24.0;
      A     M 21.4;
      AN    M 11.0;
      S     M 28.7;
M017: L     L#1600;
      L     DB17.DBD 170;
      +     L#1600;
      ==D;
      JC    M019;
      T     LD 0;
      A     M 24.1;
      A     M 11.1;
      R     M 11.1;
      JC    M019;
      A     M 24.1;
      AN    M 11.1;
      AN    M 21.4;
      S     M [LD 0];
      JC    M019;
      A     M 21.4;
      A     M 11.1;
      AN    M 24.1;
      JCN   M018;
      L     DB17.DBW 122;
      +     1792;
      ITD;
      T     LD 4;
      S     M [LD 4];
      R     M 11.1;
      R     M [LD 0];
      JU    M019;
M018: A     M 24.1;
      A     M 21.4;
      AN    M 11.1;
      S     M 29.0;
M019: L     L#1600;
      L     DB17.DBD 174;
      +     L#1600;
      ==D;
      JC    M021;
      T     LD 0;
      A     M 24.2;
      A     M 11.2;
      R     M 11.2;
      JC    M021;
      A     M 24.2;
      AN    M 11.2;
      AN    M 21.4;
      S     M [LD 0];
      JC    M021;
      A     M 21.4;
      A     M 11.2;
      AN    M 24.2;
      JCN   M020;
      L     DB17.DBW 124;
      +     1792;
      ITD;
      T     LD 4;
      S     M [LD 4];
      R     M 11.2;
      R     M [LD 0];
      JU    M021;
M020: A     M 24.2;
      A     M 21.4;
      AN    M 11.2;
      S     M 29.1;
M021: L     L#1600;
      L     DB17.DBD 178;
      +     L#1600;
      ==D;
      JC    M023;
      T     LD 0;
      A     M 24.3;
      A     M 11.3;
      R     M 11.3;
      JC    M023;
      A     M 24.3;
      AN    M 11.3;
      AN    M 21.4;
      S     M [LD 0];
      JC    M023;
      A     M 21.4;
      A     M 11.3;
      AN    M 24.3;
      JCN   M022;
      L     DB17.DBW 126;
      +     1792;
      ITD;
      T     LD 4;
      S     M [LD 4];
      R     M 11.3;
      R     M [LD 0];
      JU    M023;
M022: A     M 24.3;
      A     M 21.4;
      AN    M 11.3;
      S     M 29.2;
M023: L     L#1600;
      L     DB17.DBD 182;
      +     L#1600;
      ==D;
      JC    M025;
      T     LD 0;
      A     M 24.4;
      A     M 11.4;
      R     M 11.4;
      JC    M025;
      A     M 24.4;
      AN    M 11.4;
      AN    M 21.4;
      S     M [LD 0];
      JC    M025;
      A     M 21.4;
      A     M 11.4;
      AN    M 24.4;
      JCN   M024;
      L     DB17.DBW 128;
      +     1792;
      ITD;
      T     LD 4;
      S     M [LD 4];
      R     M 11.4;
      R     M [LD 0];
      JU    M025;
M024: A     M 24.4;
      A     M 21.4;
      AN    M 11.4;
      S     M 29.3;
M025: L     L#1600;
      L     DB17.DBD 186;
      +     L#1600;
      ==D;
      JC    M027;
      T     LD 0;
      A     M 24.5;
      A     M 11.5;
      R     M 11.5;
      JC    M027;
      A     M 24.5;
      AN    M 11.5;
      AN    M 21.4;
      S     M [LD 0];
      JC    M027;
      A     M 21.4;
      A     M 11.5;
      AN    M 24.5;
      JCN   M026;
      L     DB17.DBW 130;
      +     1792;
      ITD;
      T     LD 4;
      S     M [LD 4];
      R     M 11.5;
      R     M [LD 0];
      JU    M027;
M026: A     M 24.5;
      A     M 21.4;
      AN    M 11.5;
      S     M 29.4;
M027: L     L#1600;
      L     DB17.DBD 198;
      +     L#1600;
      ==D;
      JC    M029;
      T     LD 0;
      A     M 21.6;
      A     M 10.7;
      R     M 10.7;
      JC    M029;
      A     M 21.6;
      AN    M 10.7;
      AN    M 21.4;
      S     M [LD 0];
      JC    M029;
      A     M 21.4;
      A     M 10.7;
      AN    M 21.6;
      JCN   M028;
      S     M 223.4;
      R     M 10.7;
      R     M [LD 0];
      JU    M029;
M028: A     M 21.6;
      A     M 21.4;
      AN    M 10.7;
      S     M 29.7;
NETWORK
TITLE =
M029: A     M 21.5;
      S     M 200.0;
      A     M 21.4;
      JCN   M030;
      A     M 203.7;
      =     L 18.0;
      A     M 207.7;
      =     L 18.1;
      A     M 211.7;
      =     L 18.2;
      A     M 215.7;
      =     L 18.3;
      L     MD 200;
      CAD;
      SLD   1;
      CAD;
      T     MD 200;
      L     MD 204;
      CAD;
      SLD   1;
      CAD;
      T     MD 204;
      L     MD 208;
      CAD;
      SLD   1;
      CAD;
      T     MD 208;
      L     MD 212;
      CAD;
      SLD   1;
      CAD;
      T     MD 212;
      L     MD 216;
      CAD;
      SLD   1;
      CAD;
      T     MD 216;
      A     L 18.0;
      =     M 204.0;
      A     L 18.1;
      =     M 208.0;
      A     L 18.2;
      =     M 212.0;
      A     L 18.3;
      =     M 216.0;
      L     0;
      T     LB 18;
      JU    M031;
M030: A     M 25.4;
      JCN   M045;
      A     M 216.0;
      =     L 18.3;
      A     M 212.0;
      =     L 18.2;
      A     M 208.0;
      =     L 18.1;
      A     M 204.0;
      =     L 18.0;
      L     MD 216;
      CAD;
      SRD   1;
      CAD;
      T     MD 216;
      L     MD 212;
      CAD;
      SRD   1;
      CAD;
      T     MD 212;
      L     MD 208;
      CAD;
      SRD   1;
      CAD;
      T     MD 208;
      L     MD 204;
      CAD;
      SRD   1;
      CAD;
      T     MD 204;
      L     MD 200;
      CAD;
      SRD   1;
      CAD;
      T     MD 200;
      A     L 18.3;
      =     M 215.7;
      A     L 18.2;
      =     M 211.7;
      A     L 18.1;
      =     M 207.7;
      A     L 18.0;
      =     M 203.7;
      L     0;
      T     LB 18;
NETWORK
TITLE =
M031: L     L#1600;
      L     DB17.DBD 138;
      +     L#1600;
      ==D;
      JC    M032;
      T     LD 0;
      A     M [LD 0];
      AN    M 28.0;
      S     M 10.0;
      JC    M032;
      R     M 28.0;
M032: L     L#1600;
      L     DB17.DBD 142;
      +     L#1600;
      ==D;
      JC    M033;
      T     LD 0;
      A     M [LD 0];
      AN    M 28.1;
      S     M 10.1;
      JC    M033;
      R     M 28.1;
M033: L     L#1600;
      L     DB17.DBD 146;
      +     L#1600;
      ==D;
      JC    M034;
      T     LD 0;
      A     M [LD 0];
      AN    M 28.2;
      S     M 10.2;
      JC    M034;
      R     M 28.2;
M034: L     L#1600;
      L     DB17.DBD 150;
      +     L#1600;
      ==D;
      JC    M035;
      T     LD 0;
      A     M [LD 0];
      AN    M 28.3;
      S     M 10.3;
      JC    M035;
      R     M 28.3;
M035: L     L#1600;
      L     DB17.DBD 154;
      +     L#1600;
      ==D;
      JC    M036;
      T     LD 0;
      A     M [LD 0];
      AN    M 28.4;
      S     M 10.4;
      JC    M036;
      R     M 28.4;
M036: L     L#1600;
      L     DB17.DBD 158;
      +     L#1600;
      ==D;
      JC    M037;
      T     LD 0;
      A     M [LD 0];
      AN    M 28.5;
      S     M 10.5;
      JC    M037;
      R     M 28.5;
M037: L     L#1600;
      L     DB17.DBD 162;
      +     L#1600;
      ==D;
      JC    M038;
      T     LD 0;
      A     M [LD 0];
      AN    M 28.6;
      S     M 10.6;
      JC    M038;
      R     M 28.6;
M038: L     L#1600;
      L     DB17.DBD 166;
      +     L#1600;
      ==D;
      JC    M039;
      T     LD 0;
      A     M [LD 0];
      AN    M 28.7;
      S     M 11.0;
      JC    M039;
      R     M 28.7;
M039: L     L#1600;
      L     DB17.DBD 170;
      +     L#1600;
      ==D;
      JC    M040;
      T     LD 0;
      A     M [LD 0];
      AN    M 29.0;
      S     M 11.1;
      JC    M040;
      R     M 29.0;
M040: L     L#1600;
      L     DB17.DBD 174;
      +     L#1600;
      ==D;
      JC    M041;
      T     LD 0;
      A     M [LD 0];
      AN    M 29.1;
      S     M 11.2;
      JC    M041;
      R     M 29.1;
M041: L     L#1600;
      L     DB17.DBD 178;
      +     L#1600;
      ==D;
      JC    M042;
      T     LD 0;
      A     M [LD 0];
      AN    M 29.2;
      S     M 11.3;
      JC    M042;
      R     M 29.2;
M042: L     L#1600;
      L     DB17.DBD 182;
      +     L#1600;
      ==D;
      JC    M043;
      T     LD 0;
      A     M [LD 0];
      AN    M 29.3;
      S     M 11.4;
      JC    M043;
      R     M 29.3;
M043: L     L#1600;
      L     DB17.DBD 186;
      +     L#1600;
      ==D;
      JC    M044;
      T     LD 0;
      A     M [LD 0];
      AN    M 29.4;
      S     M 11.5;
      JC    M044;
      R     M 29.4;
M044: L     L#1600;
      L     DB17.DBD 198;
      +     L#1600;
      ==D;
      JC    M045;
      T     LD 0;
      A     M [LD 0];
      AN    M 29.7;
      S     M 10.7;
      JC    M045;
      R     M 29.7;
NETWORK
TITLE =
M045: L     DB17.DBW 54;
      ITD;
      +     L#1600;
      T     LD 0;
      A     M [LD 0];
      A     M 21.3;
      A     DB17.DBX 38.5;
      S     "10-Y14";
      AN    M [LD 0];
      AN    C 21;
      AN    DB17.DBX 39.1;
      O;
      AN    M [LD 0];
      A     M 21.3;
      A     DB17.DBX 39.1;
      ON    DB17.DBX 38.5;
      R     "10-Y14";
      L     QB 20;
      T     PQB 20;
      NOP   0;
NETWORK
TITLE =
      AN    C 21;
      =     M 0.7;
      AN    M [LD 0];
      A     M 21.3;
      CD    C 21;
      BLD   101;
      A     M [LD 0];
      L     C#2;
      S     C 21;
      NOP   0;
      NOP   0;
      NOP   0;
      NOP   0;
NETWORK
TITLE =
      AN    DB17.DBX 38.5;
      JC    M046;
      L     DB17.DBD 60;
      +     L#1600;
      T     LD 20;
      A     M [LD 20];
      =     L 28.0;
      A     M 21.4;
      A     M 5.3;
      S     M 222.1;
      R     M 5.3;
      A     L 28.0;
      A     M 21.4;
      S     M 5.3;
      L     DB17.DBD 60;
      +     L#1600;
      T     LD 24;
      A     M [LD 24];
      =     L 28.1;
      AN    L 28.1;
      A     M 23.4;
      S     M 222.2;
      O     "10-В30";
      O     M 241.1;
      O     "5-S230";
M046: R     M 5.3;
END_FUNCTION

FUNCTION FC 61 : VOID
AUTHOR : Stolz
NAME : Testdose
VERSION : 0.2
BEGIN
// (block stored without names or comments; labels and parameter names are numbered)
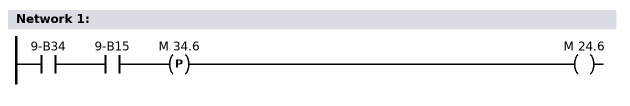
NETWORK
TITLE =
      A     "9-В34";
      A     "9-В15";
      FP    M 34.6;
      =     M 24.6;
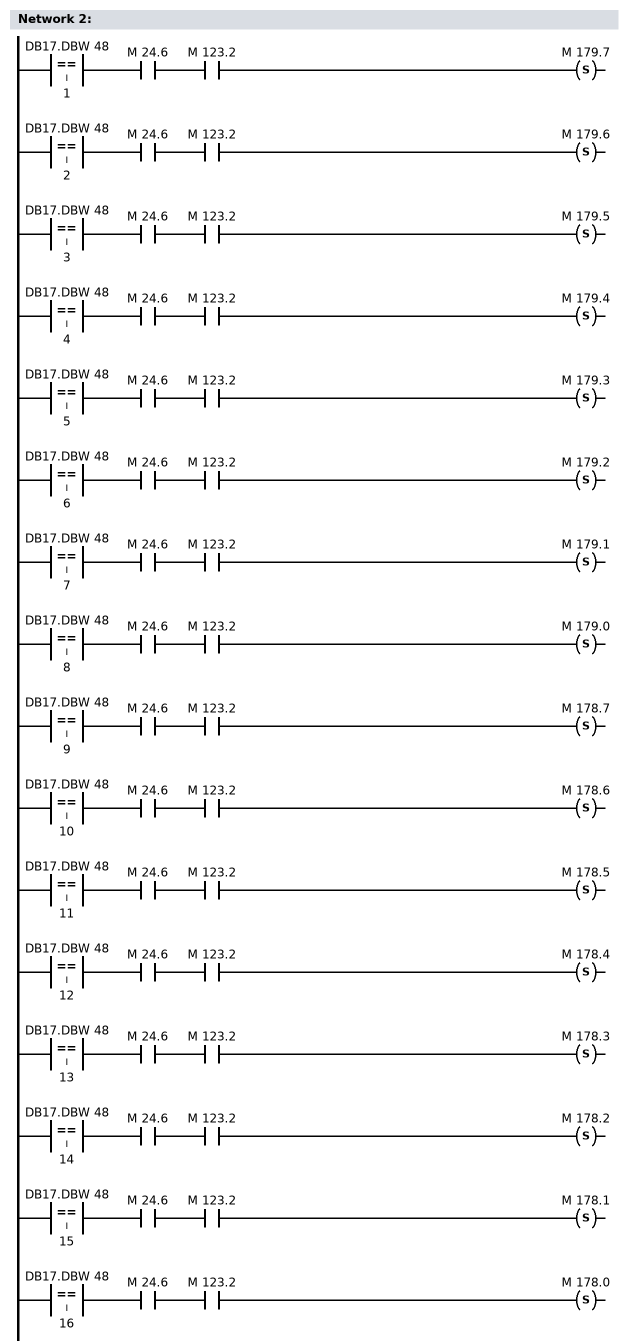
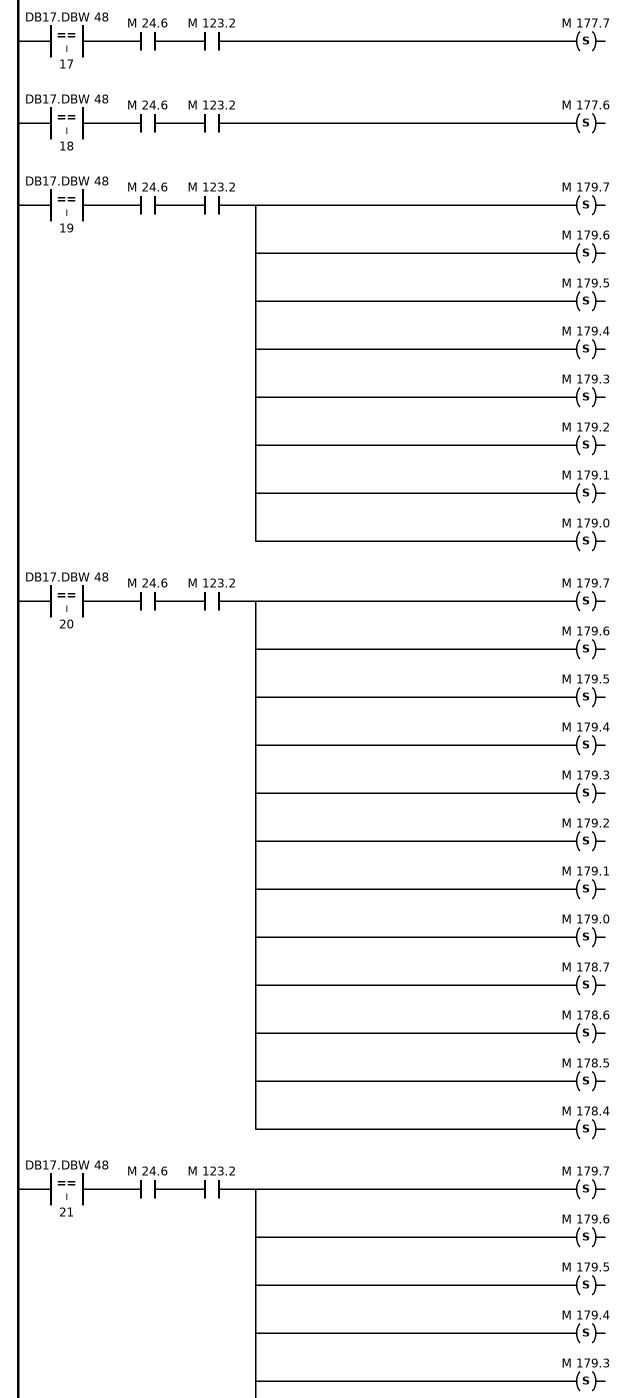
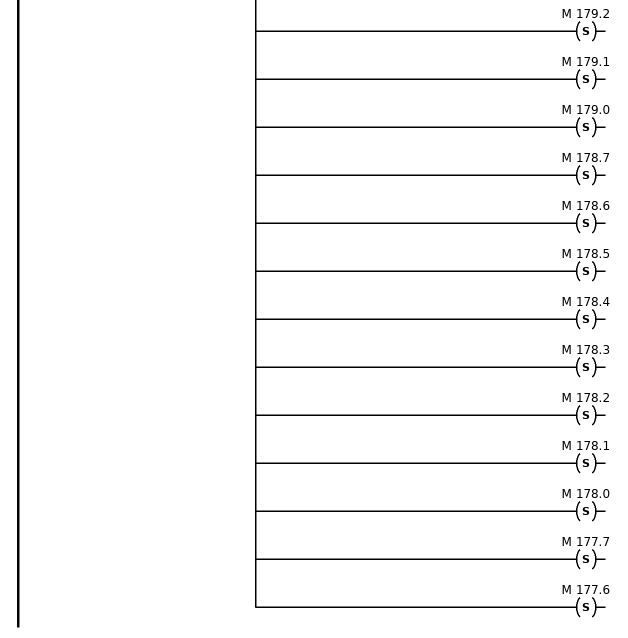
NETWORK
TITLE =
      L     DB17.DBW 48;
      L     1;
      ==I;
      A     M 24.6;
      A     M 123.2;
      S     M 179.7;
      L     DB17.DBW 48;
      L     2;
      ==I;
      A     M 24.6;
      A     M 123.2;
      S     M 179.6;
      L     DB17.DBW 48;
      L     3;
      ==I;
      A     M 24.6;
      A     M 123.2;
      S     M 179.5;
      L     DB17.DBW 48;
      L     4;
      ==I;
      A     M 24.6;
      A     M 123.2;
      S     M 179.4;
      L     DB17.DBW 48;
      L     5;
      ==I;
      A     M 24.6;
      A     M 123.2;
      S     M 179.3;
      L     DB17.DBW 48;
      L     6;
      ==I;
      A     M 24.6;
      A     M 123.2;
      S     M 179.2;
      L     DB17.DBW 48;
      L     7;
      ==I;
      A     M 24.6;
      A     M 123.2;
      S     M 179.1;
      L     DB17.DBW 48;
      L     8;
      ==I;
      A     M 24.6;
      A     M 123.2;
      S     M 179.0;
      L     DB17.DBW 48;
      L     9;
      ==I;
      A     M 24.6;
      A     M 123.2;
      S     M 178.7;
      L     DB17.DBW 48;
      L     10;
      ==I;
      A     M 24.6;
      A     M 123.2;
      S     M 178.6;
      L     DB17.DBW 48;
      L     11;
      ==I;
      A     M 24.6;
      A     M 123.2;
      S     M 178.5;
      L     DB17.DBW 48;
      L     12;
      ==I;
      A     M 24.6;
      A     M 123.2;
      S     M 178.4;
      L     DB17.DBW 48;
      L     13;
      ==I;
      A     M 24.6;
      A     M 123.2;
      S     M 178.3;
      L     DB17.DBW 48;
      L     14;
      ==I;
      A     M 24.6;
      A     M 123.2;
      S     M 178.2;
      L     DB17.DBW 48;
      L     15;
      ==I;
      A     M 24.6;
      A     M 123.2;
      S     M 178.1;
      L     DB17.DBW 48;
      L     16;
      ==I;
      A     M 24.6;
      A     M 123.2;
      S     M 178.0;
      L     DB17.DBW 48;
      L     17;
      ==I;
      A     M 24.6;
      A     M 123.2;
      S     M 177.7;
      L     DB17.DBW 48;
      L     18;
      ==I;
      A     M 24.6;
      A     M 123.2;
      S     M 177.6;
      L     DB17.DBW 48;
      L     19;
      ==I;
      A     M 24.6;
      A     M 123.2;
      S     M 179.7;
      S     M 179.6;
      S     M 179.5;
      S     M 179.4;
      S     M 179.3;
      S     M 179.2;
      S     M 179.1;
      S     M 179.0;
      L     DB17.DBW 48;
      L     20;
      ==I;
      A     M 24.6;
      A     M 123.2;
      S     M 179.7;
      S     M 179.6;
      S     M 179.5;
      S     M 179.4;
      S     M 179.3;
      S     M 179.2;
      S     M 179.1;
      S     M 179.0;
      S     M 178.7;
      S     M 178.6;
      S     M 178.5;
      S     M 178.4;
      L     DB17.DBW 48;
      L     21;
      ==I;
      A     M 24.6;
      A     M 123.2;
      S     M 179.7;
      S     M 179.6;
      S     M 179.5;
      S     M 179.4;
      S     M 179.3;
      S     M 179.2;
      S     M 179.1;
      S     M 179.0;
      S     M 178.7;
      S     M 178.6;
      S     M 178.5;
      S     M 178.4;
      S     M 178.3;
      S     M 178.2;
      S     M 178.1;
      S     M 178.0;
      S     M 177.7;
      S     M 177.6;
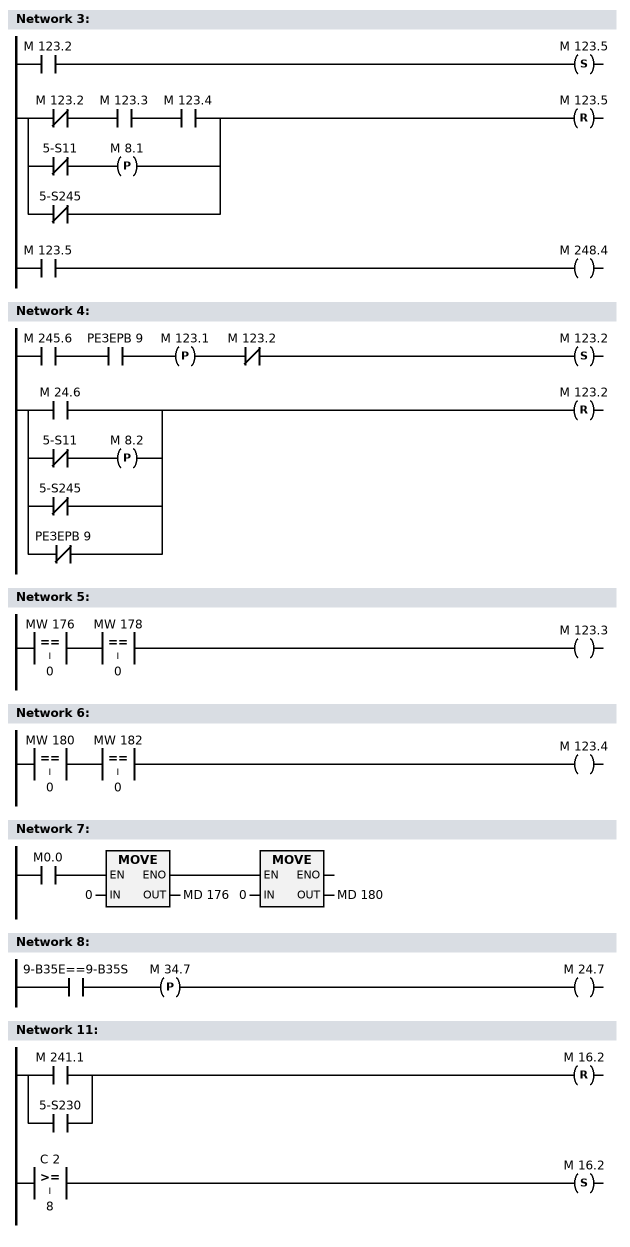
NETWORK
TITLE =
      A     M 123.2;
      S     M 123.5;
      A(;
      AN    M 123.2;
      A     M 123.3;
      A     M 123.4;
      O(;
      AN    "5-S11";
      FP    M 8.1;
      );
      ON    "5-S245";
      );
      R     M 123.5;
      A     M 123.5;
      =     M 248.4;
NETWORK
TITLE =
      A     M 245.6;
      A     "РЕЗЕРВ 9";
      FP    M 123.1;
      AN    M 123.2;
      S     M 123.2;
      A(;
      O     M 24.6;
      O(;
      AN    "5-S11";
      FP    M 8.2;
      );
      ON    "5-S245";
      ON    "РЕЗЕРВ 9";
      );
      R     M 123.2;
      NOP   0;
NETWORK
TITLE =
      A(;
      L     MW 176;
      L     0;
      ==I;
      );
      A(;
      L     MW 178;
      L     0;
      ==I;
      );
      =     M 123.3;
NETWORK
TITLE =
      A(;
      L     MW 180;
      L     0;
      ==I;
      );
      A(;
      L     MW 182;
      L     0;
      ==I;
      );
      =     M 123.4;
NETWORK
TITLE =
      A(;
      A     "М0.0";
      JNB   M001;
      L     0;
      T     MD 176;
      SET;
      SAVE;
      CLR;
M001: A     BR;
      );
      JNB   M002;
      L     0;
      T     MD 180;
M002: NOP   0;
NETWORK
TITLE =
      A     "9-В35Е==9-В35S";
      FP    M 34.7;
      =     M 24.7;
NETWORK
TITLE =
      L     DB17.DBD 2;
      +     L#1440;
      T     LD 0;
NETWORK
TITLE =
// (network holds code this reader does not know; not shown)
NETWORK
TITLE =
      O     M 241.1;
      O     "5-S230";
      R     M 16.2;
      L     C 2;
      L     8;
      >=I;
      S     M 16.2;
